(*=======================================================*)
	INIT:	(* Initialisierung *)
		st_ctrl_out.b_fehler := FALSE;
		st_ctrl_out.b_fertig := FALSE;
		st_ctrl_out.b_bereit := FALSE;
		fb_add_route_entry.bExecute := FALSE;
		fb_enum_route_entry.bExecute := FALSE;
		fb_enum_route_entry.eCmd := eEnumCmd_First;
		b_routing_station_gefunden := TRUE;
		i16_eintrag := 0;
		fb_get_local_ams_netid.bExecute := FALSE;
		fb_get_local_ams_netid.bQuit := FALSE;
		fb_get_adapters_info.bExecute := FALSE;
		fb_get_adapters_info.bQuit := FALSE;
		fb_get_host_name.bExecute := FALSE;
		fb_get_host_addr_by_name.bExecute := FALSE;
		sm_fehler_netid := FALSE;
		sm_fehler_adapter_info := FALSE;
		sm_fehler_host_name := FALSE;
		sm_fehler_host_addr := FALSE;

		FOR i16_eintrag := 0  TO (SIZEOF (arr_read_routing_info) / SIZEOF (arr_read_routing_info[0])) BY 1DO
			IF	i16_eintrag <32 THEN
				arr_read_routing_info[i16_eintrag].sName := '';
				arr_read_routing_info[i16_eintrag].sNetID := '';
				arr_read_routing_info[i16_eintrag].sAddress := '';
				arr_read_routing_info[i16_eintrag].eTransport := eRouteTransport_TCP_IP;
			END_IF
		END_FOR

		IF fb_get_local_ams_netid.bReady AND fb_get_adapters_info.bReady THEN
			fb_state_entry.i16_next_step := 20;
		END_IF

(*=======================================================*)
	20:	(* Die AMS-NetID des lokalen PC ermitteln *)
		IF fb_state_entry.E THEN
			fb_get_local_ams_netid.bExecute := TRUE;
		END_IF

		IF fb_get_local_ams_netid.bBusy THEN
			fb_get_local_ams_netid.bExecute := FALSE;
			fb_state_entry.i16_next_step := 20;
		END_IF

(*=======================================================*)
	30:
		IF NOT fb_get_local_ams_netid.bBusy  AND fb_get_local_ams_netid.bReady THEN
			IF NOT fb_get_local_ams_netid.bError THEN
				fb_state_entry.i16_next_step := 40;
			ELSE	(* Fehler *)
				sm_fehler_netid := TRUE;
				fb_state_entry.i16_next_step := 1000;
			END_IF
		END_IF

(*=======================================================*)
	40:	(* Ersten Routing Eintrag im Routingtable lesen *)
		IF fb_state_entry.E THEN
			s_temp_string_p11 := MID(fb_get_local_ams_netid.local_ams_netid, 1, 11);
			s_temp_string_p12 := MID(fb_get_local_ams_netid.local_ams_netid, 1, 12);
			s_temp_string_p13 := MID(fb_get_local_ams_netid.local_ams_netid, 1, 13);
			IF s_temp_string_p11 = '.' THEN
				(* Die vierte Zahl ist einstellig *)
				i16_temp_net_int := STRING_TO_INT(MID(fb_get_local_ams_netid.local_ams_netid, 1, 10));
			ELSIF s_temp_string_p12 = '.' THEN
				(* Die vierte Zahl ist zweistellig *)
				i16_temp_net_int := STRING_TO_INT(MID(fb_get_local_ams_netid.local_ams_netid, 2, 10));
			ELSIF s_temp_string_p13 = '.' THEN
				(* Die vierte Zahl ist dreistellig *)
				i16_temp_net_int := STRING_TO_INT(MID(fb_get_local_ams_netid.local_ams_netid, 3, 10));
			END_IF
			i16_temp_net_int := i16_temp_net_int  + 1;	(* Die NetID des Remote-Panel ist um 1 höher, als diejenige des PCs *)
			s_temp_net_string := INT_TO_STRING (i16_temp_net_int);
			s_backpanel_netid := CONCAT((CONCAT(MID(fb_get_local_ams_netid.s_ams_netid, 9, 1), s_temp_net_string)), '.1.1');
			fb_state_entry.i16_next_step := 50;
		END_IF

(*=======================================================*)
	50:	(* Die Adapter-Info des lokalen PC ermitteln *)
		IF fb_state_entry.E THEN
			fb_get_adapters_info.sNet_ID := fb_get_local_ams_netid.local_ams_netid;
			fb_get_adapters_info.bExecute := TRUE;
		END_IF

		IF fb_get_adapters_info.bBusy THEN
			fb_get_adapters_info.bExecute := FALSE;
			fb_state_entry.i16_next_step := 60;
		END_IF

(*=======================================================*)
	60:	(* Info steht zur Verfügung *)
		IF NOT fb_get_adapters_info.bBusy THEN
			IF NOT fb_get_adapters_info.bError THEN
				IF fb_get_adapters_info.bReady THEN
					st_pc_adapter_info := fb_get_adapters_info.st_ip_adapter_info;
					fb_state_entry.i16_next_step := 70;
				END_IF
			ELSE	(* Fehler *)
				sm_fehler_adapter_info := TRUE;
				fb_state_entry.i16_next_step := 1000;
			END_IF
		END_IF

(*=======================================================*)
	70:	(* Die Adapter-Info des Backpanel ermitteln *)
		IF fb_state_entry.E THEN
			fb_get_adapters_info.sNet_ID := s_backpanel_netid;
			fb_get_adapters_info.bExecute := TRUE;
		END_IF

		IF fb_get_adapters_info.bBusy THEN
			fb_get_adapters_info.bExecute := FALSE;
			fb_state_entry.i16_next_step := 80;
		END_IF

(*=======================================================*)
	80:	(* Info steht zur Verfügung *)
		IF NOT fb_get_adapters_info.bBusy THEN
			IF NOT fb_get_adapters_info.bError THEN
				IF fb_get_adapters_info.bReady THEN
					st_pc_adapter_info := fb_get_adapters_info.st_ip_adapter_info;
					s_backpanel_adresse := st_pc_adapter_info.sIpAddr;
					fb_state_entry.i16_next_step := 90;
				END_IF
			ELSE	(* Fehler *)
				sm_fehler_adapter_info := TRUE;
				fb_state_entry.i16_next_step := 1000;
			END_IF
		END_IF

(*=======================================================*)
	90:	(* Den Namen des Backpanels ermitteln *)
		IF fb_state_entry.E THEN
			fb_get_host_name.sNetID := s_backpanel_netid;
			fb_get_host_name.bExecute := TRUE;
		END_IF

		IF fb_get_host_name.bBusy THEN
			fb_get_host_name.bExecute := FALSE;
			fb_state_entry.i16_next_step := 100;
		END_IF

(*=======================================================*)
	100:	(* Info steht zur Verfügung *)
		IF NOT fb_get_host_name.bBusy THEN
			IF NOT fb_get_host_name.bError THEN
				s_backpanel_name := fb_get_host_name.sHostName;
				fb_state_entry.i16_next_step := 110;
			ELSE	(* Fehler *)
				sm_fehler_host_name := TRUE;
				fb_state_entry.i16_next_step := 1000;
			END_IF
		END_IF

(*=======================================================*)
	110:	(* Ersten Routing Eintrag im Routingtable lesen *)
		IF fb_state_entry.E THEN
			fb_enum_route_entry.bExecute := TRUE;
		END_IF

		IF fb_enum_route_entry.bBusy THEN
			fb_enum_route_entry.bExecute := FALSE;
			fb_state_entry.i16_next_step := 120;
		END_IF

(*=======================================================*)
	120:	(* Routinginformation ist vorhanden *)
		IF NOT fb_enum_route_entry.bBusy  THEN
			IF NOT fb_enum_route_entry.bError THEN
				IF NOT fb_enum_route_entry.bEOE THEN
					arr_read_routing_info[i16_eintrag] := fb_enum_route_entry.stRoute;
					fb_enum_route_entry.eCmd := eEnumCmd_Next;
					i16_eintrag := i16_eintrag + 1;
					fb_state_entry.i16_next_step := 110;
				ELSE	(* Alle vorhandenen Routingeinträge  wurden eingelesen*)
					fb_state_entry.i16_next_step := 130;
				END_IF
			ELSE	(* Fehler *)
				fb_state_entry.i16_next_step := 1000;
			END_IF
		END_IF

(*=======================================================*)
	130:	(* Alle Einträge sind gelesen *)
		IF fb_state_entry.E THEN
			(* Suche nach dem zugehörigen Backpanel *)
			FOR i16_eintrag := 0  TO (SIZEOF (arr_read_routing_info) / SIZEOF (arr_read_routing_info[0])) BY 1DO
				IF arr_read_routing_info[i16_eintrag].sNetID = s_backpanel_netid AND arr_read_routing_info[i16_eintrag].sAddress = s_backpanel_adresse THEN
					b_routing_station_gefunden := TRUE;
					fb_state_entry.i16_next_step :=  999;	(* Ende *)
					EXIT;
				ELSE
					b_routing_station_gefunden := FALSE;
				END_IF
			END_FOR
			IF NOT b_routing_station_gefunden THEN
				(* Station nicht in Liste -> eintragen *)
				fb_state_entry.i16_next_step := 140;
			END_IF
		END_IF

(*=======================================================*)
	140:	(* Routingtable mit Backpaneladresse füllen *)
		IF fb_state_entry.E THEN
			(* Initialisierung der Routingverbindung zum Backpanel *)
			fb_add_route_entry.stRoute.sName := s_backpanel_name;
			fb_add_route_entry.stRoute.sNetID := s_backpanel_netid;
			fb_add_route_entry.stRoute.sAddress := s_backpanel_adresse;
			fb_add_route_entry.stRoute.eTransport := eRouteTransport_TCP_IP;
			fb_add_route_entry.bExecute :=TRUE;
		END_IF

		IF fb_add_route_entry.bBusy THEN
			fb_add_route_entry.bExecute := FALSE;
			fb_state_entry.i16_next_step := 150;
		END_IF

(*=======================================================*)
	150:	(* Routingtable füllen läuft *)
		IF NOT fb_add_route_entry.bBusy THEN
			IF NOT fb_add_route_entry.bError THEN	(* Route wurde erfolgreich hinzugefügt *)
				fb_state_entry.i16_next_step := 999;
			ELSE	(* Fehler *)
				fb_state_entry.i16_next_step := 1000;
			END_IF
		END_IF

(*=======================================================*)
	999: (* Ende: Alle Stationen wurden im Routingtable eingetragen *)
		IF fb_r_trig_ibn_start_routing.Q THEN
			fb_state_entry.i16_next_step := INIT;
		END_IF

(*=======================================================*)
	1000: (* Fehler *)
		IF fb_state_entry.E THEN
			st_ctrl_out.b_fehler := TRUE;
			fb_ton_quitt.IN := FALSE;
			fb_add_route_entry.bExecute := FALSE;
			fb_enum_route_entry.bExecute := FALSE;
			fb_get_local_ams_netid.bExecute := FALSE;
			fb_get_local_ams_netid.bQuit := FALSE;
			fb_get_adapters_info.bExecute := FALSE;
			fb_get_adapters_info.bQuit := FALSE;
			fb_get_host_name.bExecute := FALSE;
			fb_get_host_addr_by_name.bExecute := FALSE;
		END_IF

		(*-----------------------Weiterschaltbedingungen----------------------------*)
		IF st_ctrl_in.b_quitt AND NOT fb_state_entry.E THEN
			st_ctrl_out.b_fehler := FALSE;
			fb_get_local_ams_netid .bQuit := TRUE;
			fb_get_adapters_info .bQuit := TRUE;
			fb_ton_quitt.IN := TRUE;
		END_IF

		IF fb_ton_quitt.Q OR  fb_r_trig_ibn_start_routing.Q THEN
			fb_ton_quitt.IN := FALSE;
			fb_state_entry.i16_next_step := INIT;
		END_IF
END_CASE

fb_state_entry(
	i16_next_step:= ,
	i16_pos:= 2,
	s_debugtext:= ,
	E=> ,
	X=> , 
	i16_step=> ,
	i16_last_step=> );

fb_get_local_ams_netid(
	bExecute:= , 
	bQuit:= , 
	bBusy=> , 
	bReady=> , 
	bError=> , 
	nErrId=> , 
	s_ams_netid=> );

fb_add_route_entry(
	sNetID:= '',
	stRoute:= ,
	bExecute:= ,
	tTimeout:= DEFAULT_ADS_TIMEOUT,
	bBusy=> ,
	bError=> ,
	nErrID=> );

fb_enum_route_entry(
	sNetID:= '',
	eCmd:= , 
	bExecute:= , 
	tTimeout:= DEFAULT_ADS_TIMEOUT,
	bBusy=> ,
	bError=> , 
	nErrID=> , 
	bEOE=> , 
	stRoute=> );

fb_get_adapters_info(
	sNet_ID:= , 
	bExecute:= , 
	bQuit:= , 
	bBusy=> ,
	bReady=> , 
	bError=> ,
	nErrId=> , 
	st_ip_adapter_info=> );

fb_get_host_name(
	sNetID:= ,
	bExecute:= , 
	tTimeout:= DEFAULT_ADS_TIMEOUT,
	bBusy=> , 
	bError=> ,
	nErrID=> , 
	sHostName=> );

fb_get_host_addr_by_name(
	sNetID:= '',
	sHostName:= ,
	bExecute:= , 
	tTimeout:= DEFAULT_ADS_TIMEOUT,
	bBusy=> , 
	bError=> , 
	nErrID=> , 
	sAddr=> , 
	arrAddr=> );

IF st_config.b_config_fertig THEN
	garr_stoermeldungen[st_config.i16_meld_startindex + 0] := sm_fehler_netid;
	garr_stoermeldungen[st_config.i16_meld_startindex + 1] := sm_fehler_adapter_info;
	garr_stoermeldungen[st_config.i16_meld_startindex + 2] := FALSE;
	garr_stoermeldungen[st_config.i16_meld_startindex + 3] := sm_fehler_host_addr;
	garr_stoermeldungen[st_config.i16_meld_startindex + 4] := FALSE;
	garr_stoermeldungen[st_config.i16_meld_startindex + 5] := FALSE;
	garr_stoermeldungen[st_config.i16_meld_startindex + 6] := FALSE;
	garr_stoermeldungen[st_config.i16_meld_startindex + 7] := FALSE;
	garr_stoermeldungen[st_config.i16_meld_startindex + 8] := FALSE;
	garr_stoermeldungen[st_config.i16_meld_startindex + 9] := FALSE;
	garr_stoermeldungen[st_config.i16_meld_startindex + 10] := FALSE;
	garr_stoermeldungen[st_config.i16_meld_startindex + 11] := FALSE;
	garr_stoermeldungen[st_config.i16_meld_startindex + 12] := FALSE;
	garr_stoermeldungen[st_config.i16_meld_startindex + 13] := FALSE;
	garr_stoermeldungen[st_config.i16_meld_startindex + 14] := FALSE;
	garr_stoermeldungen[st_config.i16_meld_startindex + 15] := FALSE;
	garr_stoermeldungen[st_config.i16_meld_startindex + 16] := FALSE;
	garr_stoermeldungen[st_config.i16_meld_startindex + 17] := FALSE;
	garr_stoermeldungen[st_config.i16_meld_startindex + 18] := FALSE;
	garr_stoermeldungen[st_config.i16_meld_startindex + 19] := FALSE;
	
	garr_betriebsmeldungen[st_config.i16_meld_startindex + 0] := FALSE;
	garr_betriebsmeldungen[st_config.i16_meld_startindex + 1] := FALSE;
	garr_betriebsmeldungen[st_config.i16_meld_startindex + 2] := FALSE;
	garr_betriebsmeldungen[st_config.i16_meld_startindex + 3] := FALSE;
	garr_betriebsmeldungen[st_config.i16_meld_startindex + 4] := FALSE;
	garr_betriebsmeldungen[st_config.i16_meld_startindex + 5] := FALSE;
	garr_betriebsmeldungen[st_config.i16_meld_startindex + 6] := FALSE;
	garr_betriebsmeldungen[st_config.i16_meld_startindex + 7] := FALSE;
	garr_betriebsmeldungen[st_config.i16_meld_startindex + 8] := FALSE;
	garr_betriebsmeldungen[st_config.i16_meld_startindex + 9] := FALSE;
	garr_betriebsmeldungen[st_config.i16_meld_startindex + 10] := FALSE;
	garr_betriebsmeldungen[st_config.i16_meld_startindex + 11] := FALSE;
	garr_betriebsmeldungen[st_config.i16_meld_startindex + 12] := FALSE;
	garr_betriebsmeldungen[st_config.i16_meld_startindex + 13] := FALSE;
	garr_betriebsmeldungen[st_config.i16_meld_startindex + 14] := FALSE;
	garr_betriebsmeldungen[st_config.i16_meld_startindex + 15] := FALSE;
	garr_betriebsmeldungen[st_config.i16_meld_startindex + 16] := FALSE;
	garr_betriebsmeldungen[st_config.i16_meld_startindex + 17] := FALSE;
	garr_betriebsmeldungen[st_config.i16_meld_startindex + 18] := FALSE;
	garr_betriebsmeldungen[st_config.i16_meld_startindex + 19] := FALSE;
END_IF
END_PROGRAM

(* POU EPT Lib/Programmbausteine/Routing/ST_GetAdaptersInfo, ST *)
FUNCTION_BLOCK ST_GetAdaptersInfo
VAR_INPUT
	sNet_ID						: T_AmsNetId;
	bExecute					: BOOL;
	bQuit						: BOOL;
END_VAR
VAR_OUTPUT
	bBusy						: BOOL;
	bReady						: BOOL;
	bError						: BOOL;
	nErrId						: UDINT;
	st_ip_adapter_info				: ST_IpAdapterInfo;
END_VAR
VAR
	fb_ton_quitt					: TON;
	fb_state_entry					: ST_StateEntry;
	fb_r_trig_execute				: R_TRIG;
	fb_get_adapters_info			: FB_GetAdaptersInfo;
	arr_adapters 					: ARRAY[0..MAX_LOCAL_ADAPTERS] OF ST_IpAdapterInfo;
END_VAR
(* Auslesen von IP-Adresse usw. des lokalen PCs *)
fb_r_trig_execute(CLK:= bExecute, Q=> );
fb_ton_quitt(IN:= , PT:= t#100ms, Q=> , ET=> );

(* =======================================Toplevel========================================== *)
IF fb_state_entry.i16_next_step > INIT AND fb_state_entry.i16_next_step < FEHLER THEN
	 IF fb_get_adapters_info.bError THEN
		fb_state_entry.i16_next_step := FEHLER;
	END_IF
END_IF

fb_state_entry(
	i16_next_step:= ,
	i16_pos:= 1,
	s_debugtext:= ,
	E=> ,
	X=> ,
	i16_step=> ,
	i16_last_step=> );

CASE fb_state_entry.i16_step OF
(*=======================================================*)
	0:
		fb_state_entry.i16_next_step := INIT;

(*=======================================================*)
	INIT:(* INIT *)
		bBusy := FALSE;
		bReady := FALSE;
		bError := FALSE;
		nErrId := 0;
		fb_get_adapters_info.bExecute := FALSE;
		fb_state_entry.i16_next_step := 20;

(*=======================================================*)
	20:	(* Warte auf Execute-Befehl *)
		IF fb_state_entry.E THEN
			bReady := TRUE;
		END_IF

		(*-----------------------Weiterschaltbedingungen----------------------------*)
		IF fb_r_trig_execute.Q THEN
			bReady := FALSE;
			bBusy := TRUE;
			fb_state_entry.i16_next_step := 30;
		END_IF

(*=======================================================*)
	30:	(* Starte mit Auslesen der Adapter-Info des lokalen PC *)
		IF fb_state_entry.E THEN
			fb_get_adapters_info.bExecute := TRUE;
		END_IF

		IF fb_get_adapters_info.bBusy THEN
			fb_get_adapters_info.bExecute := FALSE;
			fb_state_entry.i16_next_step := 40;
		END_IF

(*=======================================================*)
	40:	(* Adapter-Info wurde ausgelesen *)
		IF NOT fb_get_adapters_info.bBusy THEN
			IF NOT fb_get_adapters_info.bError THEN
				bBusy := FALSE;
				fb_state_entry.i16_next_step := 999;
			ELSE	(* Fehler *)
				fb_state_entry.i16_next_step := 1000;
			END_IF
		END_IF

(*=======================================================*)
	999:	(* Fertig *)
		st_ip_adapter_info := arr_adapters[1];
		fb_state_entry.i16_next_step := 20;

(*=======================================================*)
	FEHLER: (* Fehler *)
		IF fb_state_entry.E THEN
			bBusy := FALSE;
			bReady := FALSE;
			bError := TRUE;
			fb_get_adapters_info.bExecute := FALSE;
			fb_ton_quitt.IN := FALSE;
		END_IF

		(*-----------------------Weiterschaltbedingungen----------------------------*)
		IF bQuit AND NOT fb_state_entry.E THEN
			bError := FALSE;
			fb_ton_quitt.IN := TRUE;
			(* Quittierflanke für FB *)
			fb_get_adapters_info.bExecute := TRUE;
		END_IF

		IF fb_ton_quitt.Q THEN
			fb_ton_quitt.IN := FALSE;
			fb_state_entry.i16_next_step := INIT;
		END_IF
END_CASE

fb_state_entry(
	i16_next_step:= , 
	i16_pos:= 2,
	s_debugtext:= ,
	E=> ,
	X=> ,
	i16_step=> ,
	i16_last_step=> );

fb_get_adapters_info(
	sNetID:= sNet_ID,
	bExecute:= , 
	tTimeout:= DEFAULT_ADS_TIMEOUT,
	bBusy=> ,
	bError=> , 
	nErrID=> nErrId,
	arrAdapters=> arr_adapters,
	nCount=> , 
	nGet=> );
END_FUNCTION_BLOCK

(* POU EPT Lib/Programmbausteine/Routing/PC-Suche/ST_RoutingNachbarPC, ST *)
PROGRAM ST_RoutingNachbarPC
VAR_INPUT
	st_config						: struct_config;
	st_ctrl_in						: struct_ctrl_in;
END_VAR
VAR_OUTPUT
	st_ctrl_out					: struct_ctrl_out;
END_VAR
VAR
	arr_read_routing_info			: ARRAY [0..31] OF ST_AmsRouteEntry;
	fb_add_route_entry			: FB_AddRouteEntry;
	fb_enum_route_entry			: FB_EnumRouteEntry;
	fb_ton_quitt					: TON;
	fb_state_entry					: ST_StateEntry;
	i16_geschriebene_eintraege	: INT := 0;
	i16_vorhandene_eintraege		: INT := 0;
	b_ibn_start_routing			: BOOL := FALSE;
	fb_r_trig_ibn_start_routing		: R_TRIG;
	fb_ton_ibn_start_routing		: TON;
	sm_fehler_remotesuche		: BOOL := FALSE;
	sm_fehler_netid				: BOOL := FALSE;
	fb_suche_remote_pc			: ST_SucheRemotePC;
	fb_get_local_ams_netid		: ST_GetLocalAMSNetID;
	i16_eintrag					: INT := 0;
END_VAR
fb_ton_quitt(IN:= , PT:= t#100ms, Q=> , ET=> );
fb_r_trig_ibn_start_routing(CLK:= b_ibn_start_routing, Q=> );
fb_ton_ibn_start_routing(IN:= , PT:= t#1s, Q=> , ET=> );

IF fb_r_trig_ibn_start_routing.Q THEN
	fb_ton_ibn_start_routing.IN := TRUE;
ELSE
	IF fb_ton_ibn_start_routing.Q THEN
		b_ibn_start_routing := FALSE;
	 	fb_ton_ibn_start_routing.IN := FALSE;
	END_IF
END_IF

fb_state_entry(
	i16_next_step:= ,
	i16_pos:= 1,
	s_debugtext:= ,
	E=> ,
	X=> ,
	i16_step=> ,
	i16_last_step=> );

CASE fb_state_entry.i16_step OF
(*=======================================================*)
	0:	(* Initialisierung *)
		st_ctrl_out.b_fehler := TRUE;
		st_ctrl_out.b_bereit := TRUE;
		st_ctrl_out.b_fertig := TRUE;
		fb_add_route_entry.bExecute := FALSE;
		fb_enum_route_entry.bExecute := FALSE;
		fb_suche_remote_pc.bQuit := FALSE;
		fb_suche_remote_pc.bExecute := FALSE;
		fb_get_local_ams_netid .bQuit := FALSE;
		fb_get_local_ams_netid.bExecute := FALSE;
		fb_enum_route_entry.eCmd := eEnumCmd_First;
		i16_geschriebene_eintraege := 0;
		i16_vorhandene_eintraege := 0;
		sm_fehler_remotesuche := FALSE;
		sm_fehler_netid := FALSE;

		FOR i16_eintrag := 0  TO (SIZEOF (arr_read_routing_info) / SIZEOF (arr_read_routing_info[0])) BY 1DO
			arr_read_routing_info[i16_eintrag].sName := '';
			arr_read_routing_info[i16_eintrag].sNetID := '';
			arr_read_routing_info[i16_eintrag].sAddress := '';
			arr_read_routing_info[i16_eintrag].eTransport := eRouteTransport_TCP_IP;
		END_FOR

		fb_state_entry.i16_next_step := 10;

(*=======================================================*)
	10:	(* Die AMS-NetID des lokalen PC ermitteln *)
		IF fb_state_entry.E THEN
			fb_get_local_ams_netid.bExecute := TRUE;
		END_IF

		IF fb_get_local_ams_netid.bBusy THEN
			fb_get_local_ams_netid.bExecute := FALSE;
			fb_state_entry.i16_next_step := 20;
		END_IF

(*=======================================================*)
	20:
		IF NOT fb_get_local_ams_netid.bBusy  THEN
			IF NOT fb_get_local_ams_netid.bError THEN
				fb_state_entry.i16_next_step := 100;
			ELSE	(* Fehler *)
				sm_fehler_netid := TRUE;
				fb_state_entry.i16_next_step := 1000;
			END_IF
		END_IF

(*=======================================================*)
	100:	(* Ersten Routing Eintrag im Routingtable lesen *)
		IF fb_state_entry.E THEN
			fb_enum_route_entry.bExecute := TRUE;
		END_IF

		IF fb_enum_route_entry.bBusy THEN
			fb_enum_route_entry.bExecute := FALSE;
			fb_state_entry.i16_next_step := 110;
		END_IF

(*=======================================================*)
	110:	(* Routinginformation ist vorhanden *)
		IF NOT fb_enum_route_entry.bBusy  THEN
			IF NOT fb_enum_route_entry.bError THEN
				IF NOT fb_enum_route_entry.bEOE THEN
					arr_read_routing_info[i16_vorhandene_eintraege] := fb_enum_route_entry.stRoute;
					fb_enum_route_entry.eCmd := eEnumCmd_Next;
					fb_state_entry.i16_next_step := 120;
				ELSE	(* Alle vorhandenen Routingeinträge  wurden eingelesen*)
					fb_state_entry.i16_next_step := 130;
				END_IF
			ELSE	(* Fehler *)
				fb_state_entry.i16_next_step := 1000;
			END_IF
		END_IF

(*=======================================================*)
	120:	(* Zähler erhöhen *)
		IF fb_state_entry.E THEN
			i16_vorhandene_eintraege := i16_vorhandene_eintraege + 1;
		END_IF

		fb_state_entry.i16_next_step := 100;

(*=======================================================*)
	130:	(* Suche Nachbar-PCs im Maschinennetz *)
		IF fb_state_entry.E THEN
			fb_suche_remote_pc.bExecute := TRUE;
		END_IF

		IF fb_suche_remote_pc.bBusy THEN
			fb_suche_remote_pc.bExecute := FALSE;
			fb_state_entry.i16_next_step := 140;
		END_IF

(*=======================================================*)
	140:	(* Suchvorgang und beendet *)
		IF NOT fb_suche_remote_pc.bBusy  THEN
			IF NOT fb_suche_remote_pc.bError THEN
				fb_state_entry.i16_next_step := 150;
			ELSE	(* Fehler *)
				sm_fehler_remotesuche := TRUE;
				fb_state_entry.i16_next_step := 1000;
			END_IF
		END_IF

(*=======================================================*)
	150:	(* Die Route der gefundenen Nachbar-PCs eintragen *)
		IF fb_state_entry.E THEN
			fb_add_route_entry.stRoute.sName := fb_suche_remote_pc.st_remote_pcinfo_struct[i16_geschriebene_eintraege].Name;
			fb_add_route_entry.stRoute.sNetID := fb_suche_remote_pc.st_remote_pcinfo_struct[i16_geschriebene_eintraege].NetId;
			fb_add_route_entry.stRoute.sAddress := DELETE(fb_add_route_entry.stRoute.sNetID, 4, 12);
			fb_add_route_entry.stRoute.eTransport := eRouteTransport_TCP_IP;
			fb_add_route_entry.bExecute :=TRUE;
			i16_geschriebene_eintraege := i16_geschriebene_eintraege + 1;
		END_IF

		IF fb_add_route_entry.bBusy THEN
			fb_add_route_entry.bExecute := FALSE;
			fb_state_entry.i16_next_step := 160;
		END_IF

(*=======================================================*)
	160:	(* Routingtable füllen läuft *)
		IF NOT fb_add_route_entry.bBusy THEN
			IF NOT fb_add_route_entry.bError THEN	(* Route wurde erfolgreich hinzugefügt *)
				(* Routingtable mit fehlenden Stationsadressen füllen wenn notwendig *)
				IF i16_geschriebene_eintraege < i16_vorhandene_eintraege THEN
					fb_state_entry.i16_next_step := 150;
				ELSE
					fb_state_entry.i16_next_step := 999;
				END_IF
			ELSE	(* Fehler *)
				fb_state_entry.i16_next_step := 1000;
			END_IF
		END_IF

(*=======================================================*)
	999: (* Ende: Alle Stationen wurden im Routingtable eingetragen *)
		IF fb_state_entry.E THEN
			st_ctrl_out.b_fertig := TRUE;
		END_IF

(*=======================================================*)
	1000: (* Fehler *)
		IF fb_state_entry.E THEN
			st_ctrl_out.b_fehler := TRUE;
			fb_ton_quitt.IN := FALSE;
			fb_add_route_entry.bExecute := FALSE;
			fb_enum_route_entry.bExecute := FALSE;
			fb_suche_remote_pc.bExecute := FALSE;
			fb_suche_remote_pc.bQuit := FALSE;
			fb_get_local_ams_netid.bExecute := FALSE;
			fb_get_local_ams_netid.bQuit := FALSE;
		END_IF

		(*-----------------------Weiterschaltbedingungen----------------------------*)
		IF st_ctrl_in.b_quitt AND NOT fb_state_entry.E THEN
			st_ctrl_out.b_fehler := FALSE;
			fb_ton_quitt.IN := TRUE;
			fb_suche_remote_pc.bQuit := TRUE;
			fb_get_local_ams_netid .bQuit := TRUE;
		END_IF

		IF fb_ton_quitt.Q OR  fb_r_trig_ibn_start_routing.Q THEN
			fb_ton_quitt.IN := FALSE;
			fb_state_entry.i16_next_step := 0;
		END_IF
END_CASE

fb_state_entry(
	i16_next_step:= , 
	i16_pos:= 2,
	s_debugtext:= ,
	E=> ,
	X=> , 
	i16_step=> ,
	i16_last_step=> );

fb_get_local_ams_netid(
	bExecute:= , 
	bQuit:= , 
	bBusy=> , 
	bReady=> , 
	bError=> , 
	nErrId=> , 
	s_ams_netid=> );

fb_suche_remote_pc(
	bExecute:= ,
	bQuit:= , 
	bBusy=> , 
	bError=> , 
	nErrId=> );

fb_add_route_entry(
	sNetID:= ,
	stRoute:= ,
	bExecute:= ,
	tTimeout:= DEFAULT_ADS_TIMEOUT,
	bBusy=> , 
	bError=> , 
	nErrID=> );

fb_enum_route_entry(
	sNetID:= ,
	eCmd:= , 
	bExecute:= , 
	tTimeout:= DEFAULT_ADS_TIMEOUT,
	bBusy=> , 
	bError=> , 
	nErrID=> , 
	bEOE=> , 
	stRoute=> );

IF st_config.b_config_fertig THEN
	garr_stoermeldungen[st_config.i16_meld_startindex + 0] := sm_fehler_remotesuche;
	garr_stoermeldungen[st_config.i16_meld_startindex + 1] := sm_fehler_netid;
	garr_stoermeldungen[st_config.i16_meld_startindex + 2] := FALSE;
	garr_stoermeldungen[st_config.i16_meld_startindex + 3] := FALSE;
	garr_stoermeldungen[st_config.i16_meld_startindex + 4] := FALSE;
	garr_stoermeldungen[st_config.i16_meld_startindex + 5] := FALSE;
	garr_stoermeldungen[st_config.i16_meld_startindex + 6] := FALSE;
	garr_stoermeldungen[st_config.i16_meld_startindex + 7] := FALSE;
	garr_stoermeldungen[st_config.i16_meld_startindex + 8] := FALSE;
	garr_stoermeldungen[st_config.i16_meld_startindex + 9] := FALSE;
	garr_stoermeldungen[st_config.i16_meld_startindex + 10] := FALSE;
	garr_stoermeldungen[st_config.i16_meld_startindex + 11] := FALSE;
	garr_stoermeldungen[st_config.i16_meld_startindex + 12] := FALSE;
	garr_stoermeldungen[st_config.i16_meld_startindex + 13] := FALSE;
	garr_stoermeldungen[st_config.i16_meld_startindex + 14] := FALSE;
	garr_stoermeldungen[st_config.i16_meld_startindex + 15] := FALSE;
	garr_stoermeldungen[st_config.i16_meld_startindex + 16] := FALSE;
	garr_stoermeldungen[st_config.i16_meld_startindex + 17] := FALSE;
	garr_stoermeldungen[st_config.i16_meld_startindex + 18] := FALSE;
	garr_stoermeldungen[st_config.i16_meld_startindex + 19] := FALSE;
	
	garr_betriebsmeldungen[st_config.i16_meld_startindex + 0] := FALSE;
	garr_betriebsmeldungen[st_config.i16_meld_startindex + 1] := FALSE;
	garr_betriebsmeldungen[st_config.i16_meld_startindex + 2] := FALSE;
	garr_betriebsmeldungen[st_config.i16_meld_startindex + 3] := FALSE;
	garr_betriebsmeldungen[st_config.i16_meld_startindex + 4] := FALSE;
	garr_betriebsmeldungen[st_config.i16_meld_startindex + 5] := FALSE;
	garr_betriebsmeldungen[st_config.i16_meld_startindex + 6] := FALSE;
	garr_betriebsmeldungen[st_config.i16_meld_startindex + 7] := FALSE;
	garr_betriebsmeldungen[st_config.i16_meld_startindex + 8] := FALSE;
	garr_betriebsmeldungen[st_config.i16_meld_startindex + 9] := FALSE;
	garr_betriebsmeldungen[st_config.i16_meld_startindex + 10] := FALSE;
	garr_betriebsmeldungen[st_config.i16_meld_startindex + 11] := FALSE;
	garr_betriebsmeldungen[st_config.i16_meld_startindex + 12] := FALSE;
	garr_betriebsmeldungen[st_config.i16_meld_startindex + 13] := FALSE;
	garr_betriebsmeldungen[st_config.i16_meld_startindex + 14] := FALSE;
	garr_betriebsmeldungen[st_config.i16_meld_startindex + 15] := FALSE;
	garr_betriebsmeldungen[st_config.i16_meld_startindex + 16] := FALSE;
	garr_betriebsmeldungen[st_config.i16_meld_startindex + 17] := FALSE;
	garr_betriebsmeldungen[st_config.i16_meld_startindex + 18] := FALSE;
	garr_betriebsmeldungen[st_config.i16_meld_startindex + 19] := FALSE;
END_IF
END_PROGRAM

(* POU EPT Lib/Programmbausteine/Routing/PC-Suche/ST_SucheRemotePC, ST *)
FUNCTION_BLOCK ST_SucheRemotePC
VAR_INPUT
	bExecute			: BOOL;
	bQuit				: BOOL;
END_VAR
VAR_OUTPUT
	bBusy				: BOOL;
	bError				: BOOL;
	nErrId				: UDINT;
END_VAR
VAR
	fb_ton_quitt					: TON;
	fb_state_entry					: ST_StateEntry;
	fb_r_trig_execute				: R_TRIG;
	i							: INT := 0;
	b_ibn_start					: BOOL := FALSE;
	fb_r_trig_ibn_start				: R_TRIG;
	fb_ton_ibn_start				: TON;
	fb_get_remote_pcinfo			:GetRemotePCInfo;
	st_remote_pcinfo_struct		:REMOTEPCINFOSTRUCT;
							       (*TYPE REMOTEPCINFOSTRUCT
									ARRAY[0..99] OF REMOTEPC;
								END_TYPE*)
							      (*TYPE REMOTEPC
								STRUCT
									NetId 	: T_AmsNetId;
									Name 	: STRING(31);
								END_STRUCT
								END_TYPE*)
END_VAR
fb_r_trig_execute(CLK:= bExecute, Q=> );
fb_ton_quitt(IN:= , PT:= t#100ms, Q=> , ET=> );

fb_r_trig_ibn_start(CLK:= b_ibn_start, Q=> );
fb_ton_ibn_start(IN:= , PT:= t#1s, Q=> , ET=> );

IF fb_r_trig_ibn_start.Q THEN
	fb_ton_ibn_start.IN := TRUE;
ELSE
	IF fb_ton_ibn_start.Q THEN
		b_ibn_start := FALSE;
	 	fb_ton_ibn_start.IN := FALSE;
	END_IF
END_IF

fb_state_entry(
	i16_next_step:= ,
	i16_pos:= 1,
	s_debugtext:= ,
	E=> ,
	X=> , 
	i16_step=> ,
	i16_last_step=> );

CASE fb_state_entry.i16_step OF
(*=======================================================*)
	0:(* INIT *)
		bBusy := FALSE;
		bError := FALSE;
		nErrId := 0;
		fb_get_remote_pcinfo.START := FALSE;
		fb_state_entry.i16_next_step := 10;

(*=======================================================*)
	10:	(* Warte auf Execute-Befehl *)
		IF fb_state_entry.E THEN
			bBusy := FALSE;
		END_IF

		IF fb_r_trig_execute.Q OR fb_r_trig_ibn_start.Q THEN
			bBusy := TRUE;
			fb_state_entry.i16_next_step := 100;
		END_IF

(*=======================================================*)
	100:	(* Starte mit Auslesen der über ADS verbundenen Nachbar-PCs *)
		IF fb_state_entry.E THEN
			fb_get_remote_pcinfo.START := TRUE;
		END_IF

		IF fb_get_remote_pcinfo.BUSY THEN
			fb_get_remote_pcinfo.START := FALSE;
			fb_state_entry.i16_next_step := 110;
		END_IF

(*=======================================================*)
	110:	(* Routinginformation über die Nachbar-PCs ist vorhanden *)
		IF NOT fb_get_remote_pcinfo.BUSY  THEN
			IF NOT fb_get_remote_pcinfo.ERR THEN
				fb_state_entry.i16_next_step := 999;
			ELSE	(* Fehler *)
				fb_state_entry.i16_next_step := 1000;
			END_IF
		END_IF

(*=======================================================*)
	999:	(* Kontrollschritt: Nachbar-PC ist gefunden *)
		fb_state_entry.i16_next_step := 10;

(*=======================================================*)
	1000: (* Fehler *)
		IF fb_state_entry.E THEN
			bBusy := FALSE;
			bError := TRUE;
			fb_ton_quitt.IN := FALSE;
		END_IF

		(*-----------------------Weiterschaltbedingungen----------------------------*)
		IF bQuit AND NOT fb_state_entry.E THEN
			bError := FALSE;
			fb_ton_quitt.IN := TRUE;
		END_IF

		IF fb_ton_quitt.Q THEN
			fb_ton_quitt.IN := FALSE;
			fb_state_entry.i16_next_step := 0;
		END_IF
END_CASE

fb_state_entry(
	i16_next_step:= , 
	i16_pos:= 2,
	s_debugtext:= ,
	E=> ,
	X=> , 
	i16_step=> ,
	i16_last_step=> );

fb_get_remote_pcinfo(
	NETID:= , 
	START:= , 
	TMOUT:= , 
	BUSY=> , 
	ERR=> , 
	ERRID=> , 
	RemotePCInfo=> st_remote_pcinfo_struct);
END_FUNCTION_BLOCK

(* POU EPT Lib/Programmbausteine/ST_start_OSK, ST *)
PROGRAM ST_start_OSK
VAR_INPUT
	bExecute			: BOOL;
END_VAR
VAR
	NT_StartProcess 		:NT_StartProcess;
	b_Start				:BOOL;

	fb_ton_start			:TON;
	fb_r_trig_start			: R_TRIG;

END_VAR
(*Windows Tastatur starten mit der Quttiertaste*)
fb_ton_start(
	IN:=bExecute,
	PT:= t#2s,);

fb_r_trig_start(
	CLK:=fb_ton_start.Q ,
	Q=> b_Start);

NT_StartProcess(
	NETID:='',
	PATHSTR	:='C:\Windows\System32\cmd.exe',
	DIRNAME	:= ,
	COMNDLINE	:='/C C:\WINDOWS\system32\taskkill /f /im osk.exe /t & start /b osk /MAX',
	START		:=b_Start,
	TMOUT		:=T#10s);

IF	NOT NT_StartProcess.BUSY AND b_Start THEN
	b_Start:=FALSE;
END_IF
END_PROGRAM

(* POU EPT Lib/Programmbausteine/ST_System_DateAndTime, ST *)
PROGRAM ST_System_DateAndTime
VAR
	w_year					: WORD := 16#0000;
	w_month					: WORD := 16#0000;
	w_day					: WORD := 16#0000;
	w_hour					: WORD := 16#0000;
	w_min					: WORD := 16#0000;
	w_sec					: WORD := 16#0000;
	fb_get_system_time 		: FB_LocalSystemTime;
END_VAR
(* =====Erzeugen der Systemzeit für die ganze Maschine======== *)
(* Die Umstellung von Sommer auf Winterzeit und umgekehrt erfolgt automatisch über die PC-Zeit *)
fb_get_system_time ( sNetID := '',
					bEnable 	:= TRUE,
					dwCycle 	:= 1,
					dwOpt	:= 1,
					tTimeout 	:= DEFAULT_ADS_TIMEOUT,
					bValid => b_system_time_valid,
					systemTime => gst_system_time, (* Systemzeit *)
					tzID 	=> );
(*=======================================================*)
gdt_system_time := SYSTEMTIME_TO_DT(fb_get_system_time.systemTime);

w_year:=gst_system_time.wYear;
w_month:=gst_system_time.wMonth;
w_day:=gst_system_time.wDay;
w_hour:=gst_system_time.wHour;
w_min:=gst_system_time.wMinute;
w_sec:=gst_system_time.wSecond;

gstr_system_time := '';
gstr_datum := '';
IF w_day < 10 THEN
	gstr_datum := CONCAT(gstr_datum ,WORD_TO_STRING(0));
END_IF;
gstr_datum := CONCAT(gstr_datum ,WORD_TO_STRING(w_day));
gstr_datum := CONCAT(gstr_datum , '.');

IF w_month < 10 THEN
	gstr_datum := CONCAT(gstr_datum ,WORD_TO_STRING(0));
END_IF;
gstr_datum := CONCAT(gstr_datum ,WORD_TO_STRING(w_month));
gstr_datum := CONCAT(gstr_datum , '.');
gstr_datum := CONCAT(gstr_datum ,WORD_TO_STRING(w_year));	(* Datum steht zur Verfügung *)

gstr_uhrzeit := '';
IF w_hour < 10 THEN
	gstr_uhrzeit := CONCAT(gstr_uhrzeit ,WORD_TO_STRING(0));
END_IF;
gstr_uhrzeit := CONCAT(gstr_uhrzeit ,WORD_TO_STRING(w_hour));
gstr_uhrzeit := CONCAT(gstr_uhrzeit , ':');

IF w_min < 10 THEN
	gstr_uhrzeit := CONCAT(gstr_uhrzeit ,WORD_TO_STRING(0));
END_IF;
gstr_uhrzeit := CONCAT(gstr_uhrzeit ,WORD_TO_STRING(w_min));
gstr_uhrzeit := CONCAT(gstr_uhrzeit , ':');

IF w_sec < 10 THEN
	gstr_uhrzeit := CONCAT(gstr_uhrzeit ,WORD_TO_STRING(0));
END_IF;
gstr_uhrzeit := CONCAT(gstr_uhrzeit ,WORD_TO_STRING(w_sec));	(* Uhrzeit steht zur Verfügung *)

gstr_system_time := CONCAT(gstr_system_time, gstr_datum );
gstr_system_time := CONCAT(gstr_system_time , ' ');
gstr_system_time := CONCAT(gstr_system_time , gstr_uhrzeit);	(* Ausgabe von Datum und Uhrzeit als String für z.B . die Visu *)
END_PROGRAM

(* POU EPT Lib/Programmbausteine/ST_UPS, ST *)
PROGRAM ST_UPS
VAR_INPUT
	st_config				: struct_config;
	st_ctrl_in				: struct_ctrl_in;
	b_Ups					: BOOL;
END_VAR
VAR_IN_OUT

END_VAR
VAR_OUTPUT
	st_ctrl_out			: struct_ctrl_out;
END_VAR
VAR
	fb_ton_quitt			: TON;
	fb_ton_uez			: TON;
	fb_state_entry			: ST_StateEntry;

	nLastErrID			:UDINT;

	fbGetUpsStatus		: FB_GetUPSStatus;

	bm_ReplaceBattery 	: BOOL;
	bm_NoPower 		: BOOL;
	bm_StatusNotValid 	: BOOL;
END_VAR
(*======================================================
   ST: ST_UPS
 ------------------------------------------------------
   Auth: 	Thomas Vilgis    						 
   Date: 	21.06.2018    						     
   Rev.: 		1.0	
   Desc:		Der Baustein liest den Status des Akkupacks aus.
			Die restliche Akkulaufzeit in Minuten kann abgefragt werden.
			Wenn der Akkupack getauscht werden muss wird angezeigt.
			Wenn sich der PC im Netzbetrieb befindet wird angezeigt.
   Historie: 	1.0

 ========================================================*)

(* Zeiten *)
fb_ton_quitt(IN:= , PT:= t#100ms, Q=> , ET=> );
fb_ton_uez(IN:= , PT:= t#20s, Q=> , ET=> );

(* Flanken *)


(* Toplevel *)
IF fb_state_entry.i16_next_step > INIT AND fb_state_entry.i16_next_step < FEHLER  THEN
	IF fb_state_entry.i16_next_step < STOP THEN
		IF st_ctrl_in.b_stop THEN
			fb_state_entry.i16_next_step := STOP;
		END_IF
	END_IF
END_IF

(* ======================================Schrittkette======================================== *)
fb_state_entry(	i16_pos:= 1);

CASE fb_state_entry.i16_step OF
(*=======================================================*)
	INIT_OBJ:
		IF st_config.b_config_fertig THEN
			fb_state_entry.i16_next_step := INIT;
		END_IF

(*=======================================================*)
	INIT:
		IF fb_state_entry.E THEN
			fb_ton_quitt.IN := FALSE;
			fb_ton_uez.IN := FALSE;
			st_ctrl_out.b_fehler := FALSE;
			st_ctrl_out.b_bereit := FALSE;
			st_ctrl_out.b_fertig := FALSE;
			st_ctrl_out.b_busy := FALSE;

			bm_ReplaceBattery := FALSE;
			bm_NoPower := FALSE;
			bm_StatusNotValid := FALSE;

			fbGetUpsStatus.bEnable := FALSE;
		END_IF

		(*-----------------------Weiterschaltbedingungen----------------------------*)
		fb_state_entry.i16_next_step := BEREIT;

(*=======================================================*)
	BEREIT:
		IF fb_state_entry.E THEN
			st_ctrl_out.b_bereit := TRUE;
		END_IF

		fbGetUpsStatus.bEnable := b_Ups;
		fb_ton_uez.IN := b_Ups;

		(*-----------------------Weiterschaltbedingungen----------------------------*)
		IF b_Ups THEN
			IF fbGetUpsStatus.bValid THEN
				fb_state_entry.i16_next_step := 110;
			ELSIF fb_ton_uez.Q THEN
				bm_StatusNotValid := TRUE;
				fb_state_entry.i16_next_step := FEHLER;
			END_IF
		END_IF

		IF fb_state_entry.X THEN
			st_ctrl_out.b_bereit := FALSE;
			st_ctrl_out.b_fertig := FALSE;
			st_ctrl_out.b_busy := TRUE;
		END_IF

(*=======================================================*)
	110:	(* Evaluation *)

		(*-----------------------Weiterschaltbedingungen----------------------------*)
		IF fbGetUpsStatus.bValid THEN
			IF NOT fbGetUpsStatus.bError THEN
				CASE fbGetUpsStatus.stStatus.eBatteryStatus OF
					BatteryUnknownStatus:	(*Der Akkustatus ist unbekannt*)
						;
					BatteryOk:			(*Der Akku ist in Ordnung*)
						bm_ReplaceBattery := FALSE;
					BatteryReplace:		(*Der Akku sollte gewechselt werden*)
						bm_ReplaceBattery := TRUE;
				END_CASE

				CASE fbGetUpsStatus.stStatus.eCommStatus OF
					UpsCommUnknownStatus:	(*Kommunikationsstatus zur USV-Hardware ist unbekannt*)
						;
					UpsCommOk:		(*Kommunikation zur USV-Hardware ist hergestellt*)
						;
					UpsCommFailed:	(*Kommunikation zur USV wurde unterbrochen*)
						;
				END_CASE

				CASE fbGetUpsStatus.stStatus.ePowerStatus OF
					PowerUnknownStatus:	(*Der Status der Stromversorgung ist unbekannt*)
						;
					PowerOnLine:		(*Das Gerät befindet sich im Netzbetrieb*)
						bm_NoPower := FALSE;
					PowerOnBattery:	(*Stromausfall ist aufgetreten und das Gerät befindet sich im Akkubetrieb*)
						bm_NoPower := TRUE;
				END_CASE
			ELSE
				nLastErrID := fbGetUpsStatus.nErrId;
				fb_state_entry.i16_next_step := FEHLER;
			END_IF
		ELSE
			bm_StatusNotValid := TRUE;
			fb_state_entry.i16_next_step := FEHLER;
		END_IF

(*=======================================================*)
	STOP, FEHLER:
		IF fb_state_entry.E THEN
			st_ctrl_out.b_fehler := fb_state_entry.i16_step = FEHLER;
			st_ctrl_out.b_gestoppt := fb_state_entry.i16_step = STOP;
			fb_ton_quitt.IN := FALSE;
			fbGetUpsStatus.bEnable := FALSE;
		END_IF

		(*-----------------------Weiterschaltbedingungen----------------------------*)
		IF st_ctrl_in.b_quitt THEN
			st_ctrl_out.b_fehler := FALSE;
			fb_ton_quitt.IN := TRUE;
		END_IF
	
		IF fb_ton_quitt.Q THEN
			fb_ton_quitt.IN := FALSE;
			fb_state_entry.i16_next_step := INIT;
		END_IF

END_CASE

fb_state_entry(i16_pos:= 2 );

fbGetUpsStatus(
	sNetId:= ,	(* wenn in AmsNetId nichts drin steht, wird immer die lokale genommen*)
	nPort:= 0,
	bEnable:= ,
	bValid=> , 
	bError=> , 
	nErrId=> ,
	stStatus=> );

IF st_config.b_config_fertig THEN
	(* Fehlermeldungen und Betriebsmeldungen ab dem Startindex in die globalen Meldungsarrays schreiben *)
	garr_stoermeldungen[st_config.i16_meld_startindex + 0] := FALSE;
	garr_stoermeldungen[st_config.i16_meld_startindex + 1] := FALSE;
	garr_stoermeldungen[st_config.i16_meld_startindex + 2] := FALSE;
	garr_stoermeldungen[st_config.i16_meld_startindex + 3] := FALSE;
	garr_stoermeldungen[st_config.i16_meld_startindex + 4] := FALSE;

	garr_betriebsmeldungen[st_config.i16_meld_startindex + 0] := bm_ReplaceBattery;
	garr_betriebsmeldungen[st_config.i16_meld_startindex + 1] := bm_NoPower;
	garr_betriebsmeldungen[st_config.i16_meld_startindex + 2] := bm_StatusNotValid;
	garr_betriebsmeldungen[st_config.i16_meld_startindex + 3] := FALSE;
	garr_betriebsmeldungen[st_config.i16_meld_startindex + 4] := FALSE;
END_IF
END_PROGRAM

(* POU Gemeinsamkeiten17xx/Achsen/ST_Bestueckachse, ST *)
PROGRAM ST_Bestueckachse
VAR_INPUT
	st_config_achse						: struct_ecd_config;
	st_ctrl_in								: struct_ctrl_in;
	e_steuerung_ein						: BOOL;
	e_ba_mit_bedingungen				: BOOL;
	e_tuere_vorne_offen					: BOOL;
	e_tuere_hinten_offen					: BOOL;
END_VAR
VAR_IN_OUT
	st_visu								: struct_ecd_visu;
END_VAR
VAR_OUTPUT
	st_ctrl_out							: struct_ctrl_out;
END_VAR
VAR
	st_sm						 		: struct_ecd_meldungen;
	st_drive_cmd							: struct_ecd_cmd;
	fb_ton_wz							: TON;
	fb_ton_quitt							: TON;
	fb_ton_wz_disable						: TON;
	fb_r_trig_tippen						: R_TRIG;
	fb_f_trig_tippen						: F_TRIG;
	fb_r_trig_taste_plus					: R_TRIG;
	fb_r_trig_taste_minus					: R_TRIG;
	fb_r_trig_start							: R_TRIG;
	fb_r_trig_hand_dialog					: R_TRIG;
	fb_r_trig_nullpunkt_setzen				: R_TRIG;
	fb_axis								: ST_AxisJobCtrl_Motion;
	fb_state_entry							: ST_StateEntry;
	fb_ton_uez							: TON;
	i, j									: INT := 0;
	lr_pos_ohneverschiebung			: LREAL;
	st_geschwindigkeiten					: struct_ecd_geschwindigkeiten;
	b_hand_dialog_aktiv					: BOOL := FALSE;
	b_nullnockenmerker					: BOOL := FALSE;

	sm_fehler_initialposition_achse			: BOOL := FALSE;
	sm_keine_nocken_definiert				: BOOL := FALSE;
	sm_fehler_ot_ut						: BOOL := FALSE;

	e_referenz_sensor						AT %I* : BOOL;
	i16_torque							AT %I* : INT;

	fb_ot_ut_ueberwachung				: ST_OT_UT_Ueberwachung;

	lr_decceleration_nothalt				: LREAL;
	lr_decceleration_normal				: LREAL;
END_VAR
(* Zeiten *)
fb_ton_wz(IN:= ,PT:= , Q=>  , ET=> );
fb_ton_uez(IN:= ,	PT:= , Q=>  , ET=> );
fb_ton_quitt(IN:= , PT:= t#100ms, Q=> , ET=> );
fb_ton_wz_disable(IN:= , PT:= t#500ms, Q=> , ET=> );

(* Flanken *)
fb_r_trig_taste_plus(CLK:= ST_Euchner_Handbedienpult.b_Taste_Plus, Q=> );
fb_r_trig_taste_minus(CLK:= ST_Euchner_Handbedienpult.b_Taste_Minus, Q=> );
fb_r_trig_start(CLK:= st_ctrl_in.b_start, Q=> );
fb_r_trig_hand_dialog(CLK:= b_hand_dialog_aktiv, Q=> );
fb_r_trig_nullpunkt_setzen(CLK:= axis_bestueckachse.st_visu.b_nullpunkt_setzen, Q=> );

(* Achse steuern *)
(* Bestueckachse *)
fb_axis(
	e_referenznocken:= ,
	b_refsensor_vorhanden:= st_config_achse.b_refsensor_vorhanden,
	b_limitsensor_positiv_vorhanden:= st_config_achse.b_limitsensor_positiv_vorhanden,
	b_limitsensor_negativ_vorhanden:= st_config_achse.b_limitsensor_negativ_vorhanden,
	i16_achstyp := st_config_achse.i16_achstyp,
	st_position:= ,
	lr_override_vorgabe:= ST_TippTasten.lr_override,
	mc_richtung_modulo:= ,
	mc_richtung_velocity:= ,
	mc_referenzmodus:= ,
	mc_buffermode_axis:= ,
	ui16_soeparam_write_value:= ,
	w_idn:= ,
	i16_nc_parameter_nummer:= ,
	r_wert_nc_write_parameter:= ,
	st_vorgabe_geschwindigkeiten:= st_geschwindigkeiten,
	lr_soll_geschwindigkeit:=,
	b_bedingung_sls:= NOT e_tuere_vorne_offen OR NOT e_tuere_hinten_offen,
	st_ads_info := ,
	st_eccoe_sdo := ,
	st_masterachse:= bestueckachse,
	st_visu_axis:= st_visu,
	st_ecd_cmd:= st_drive_cmd,
	ui16_soeparam_read_value=> ,
	r_wert_nc_read_parameter=> );

IF gi16_betriebsart <> AUTO THEN
	(* Bausteinaufruf für Kontrolle der korrekten Abfolge von OT zu UT. Nicht für Automatikbetrieb geeignet, da Aufruf in der normalen Task! *)
	fb_ot_ut_ueberwachung(
		lr_achsposition:= bestueckachse.NcToPlc.ModuloActPos,
		b_error=> sm_fehler_ot_ut);
ELSE
	sm_fehler_ot_ut := FALSE;
END_IF

IF gi16_betriebsart = HAND THEN
	(* Achse mit dem Euchner Handbediengerät vorwärts und rückwärts Bewegen*)
	IF fb_r_trig_hand_dialog.Q THEN
		fb_state_entry.i16_next_step := HANDRAD;
	END_IF

	(* Button in der Oberfläche zum setzen des Nullpunktes *)
	IF fb_r_trig_nullpunkt_setzen.Q THEN
		fb_state_entry.i16_next_step :=	NULLPUNKT_SETZEN;
	END_IF
END_IF


(* =======================================Toplevel========================================== *)
(* Starte Inbetriebnahme-Sequenz *)
IF st_ctrl_in.b_gehe_step_ibn THEN
	fb_state_entry.i16_next_step := INBETRIEBNAHME;
END_IF

(* =====Achse wird disabled===== *)
IF (NOT e_steuerung_ein OR NOT e_ba_mit_bedingungen) AND bestueckachse.Status.Operational THEN
	st_drive_cmd.enu_cmd := POWER_DISABLE;
END_IF

IF fb_state_entry.i16_next_step > INIT AND fb_state_entry.i16_next_step < FEHLER THEN
	(* =====Fehler vom Achskontroller===== *)
	IF st_drive_cmd.b_job_fehler THEN
		fb_state_entry.i16_next_step := FEHLER;
	END_IF

	IF fb_state_entry.i16_next_step > 45 THEN
		(* Devicefehler *)
		IF bestueckachse.Status.Error THEN
			st_sm.b_achsfehler := TRUE;
			fb_state_entry.i16_next_step := FEHLER;
		ELSIF bestueckachse.Status.DriveDeviceError THEN
			st_sm.b_devicefehler := TRUE;
			fb_state_entry.i16_next_step := FEHLER;
		END_IF
	END_IF

	IF fb_state_entry.i16_next_step < STOP THEN
		(* =====Achse wird gestoppt===== *)
		IF st_ctrl_in.b_stop THEN
			fb_state_entry.i16_next_step := STOP;
		ELSIF fb_state_entry.i16_next_step < HALT THEN
			(* =====Achse wird angehalten===== *)
			IF st_ctrl_in.b_halt THEN
				fb_state_entry.i16_next_step := HALT;
			END_IF
		END_IF
	END_IF
END_IF

(* ======================================Schrittkette======================================== *)
fb_state_entry(
	i16_next_step:= ,
	i16_pos:= 1,
	s_debugtext:= ,
	E=> ,
	X=> ,
	i16_step=> ,
	i16_last_step=> );

CASE fb_state_entry.i16_step OF
(*=======================================================*)
	INIT_OBJ:
		IF st_config_achse.b_config_fertig THEN
			fb_state_entry.i16_next_step := 1;
		END_IF

(*=======================================================*)
	1:	(* Warte bis NetID´s der Slaves ausgelesen sind *)
		IF fb_state_entry.E THEN
			;
		END_IF

		(*-----------------------Weiterschaltbedingungen----------------------------*)
		IF ST_EthercatDiag.st_ctrl_out.b_fertig THEN
			fb_state_entry.i16_next_step := 3;
		END_IF

(*=======================================================*)
	3:	(* Spezifische NC-Achsparameter auslesen *)
		IF fb_state_entry.E THEN
			FOR i := 0  TO (SIZEOF (nockenschaltwerk_bestueckachse.fb.arr_spur) / SIZEOF (nockenschaltwerk_bestueckachse.fb.arr_spur[0])) - 1 BY 1DO
				gst_datensatz.st_wkz.nockenschaltwerk_bestueckachse.arr_nocken[i].b_camvalid := TRUE;
			END_FOR

			fb_axis.i16_nc_parameter_nummer := MaxVelocitySystem;
			st_drive_cmd.enu_cmd := READ_NC_PARAMETER;
		END_IF

		(*-----------------------Weiterschaltbedingungen----------------------------*)
		IF st_drive_cmd.enu_cmd = NO_COMMAND THEN
			st_geschwindigkeiten.lr_maximalgeschwindigkeit := fb_axis.r_wert_nc_read_parameter(* °/s *) * 60 / 360;
			st_geschwindigkeiten.lr_auto_max := st_geschwindigkeiten.lr_maximalgeschwindigkeit;
			st_geschwindigkeiten.lr_auto_min := 50;
			st_geschwindigkeiten.lr_jog := 100;
			fb_state_entry.i16_next_step := 4;
		END_IF

(*=======================================================*)
	4:	(* Spezifische NC-Achsparameter auslesen *)
		IF fb_state_entry.E THEN
			fb_axis.i16_nc_parameter_nummer := MaxAccelerationSystem;
			st_drive_cmd.enu_cmd := READ_NC_PARAMETER;
		END_IF

		(*-----------------------Weiterschaltbedingungen----------------------------*)
		IF st_drive_cmd.enu_cmd = NO_COMMAND THEN
			st_geschwindigkeiten.lr_beschleunigung := fb_axis.r_wert_nc_read_parameter;
			fb_state_entry.i16_next_step := 5;
		END_IF

(*=======================================================*)
	5:	(* Spezifische NC-Achsparameter auslesen *)
		IF fb_state_entry.E THEN
			fb_axis.i16_nc_parameter_nummer := MaxDecelerationSystem;
			st_drive_cmd.enu_cmd := READ_NC_PARAMETER;
		END_IF

		(*-----------------------Weiterschaltbedingungen----------------------------*)
		IF st_drive_cmd.enu_cmd = NO_COMMAND THEN
			st_geschwindigkeiten.lr_verzoegerung := fb_axis.r_wert_nc_read_parameter;
			lr_decceleration_normal := st_geschwindigkeiten.lr_verzoegerung;
			lr_decceleration_nothalt := 200000.0;
			fb_state_entry.i16_next_step := 6;
		END_IF

(*=======================================================*)
	6:	(* Spezifische NC-Achsparameter auslesen *)
		IF fb_state_entry.E THEN
			fb_axis.i16_nc_parameter_nummer := MaxJerk;
			st_drive_cmd.enu_cmd := READ_NC_PARAMETER;
		END_IF

		(*-----------------------Weiterschaltbedingungen----------------------------*)
		IF st_drive_cmd.enu_cmd = NO_COMMAND THEN
			st_geschwindigkeiten.lr_ruck := fb_axis.r_wert_nc_read_parameter;
			fb_state_entry.i16_next_step := 7;
		END_IF

(*=======================================================*)
	7:	(* Konfigurationen der Achse *)
		IF fb_state_entry.E THEN
			fb_axis.st_eccoe_sdo.s_ec_slave_net_id := ST_EthercatDiag.s_ec_slave_net_id[2];
			fb_axis.st_eccoe_sdo.ui16_slave_addr := st_config_achse.ui16_ethercat_adr;
		END_IF

		(*-----------------------Weiterschaltbedingungen----------------------------*)
		fb_state_entry.i16_next_step := FEHLER; (*in Fehler gehen damit die Achsen resetet werden. Sonst steigen die Achsen bei einem TC Restart aus*)

(*=======================================================*)
	INIT:
		IF fb_state_entry.E THEN
			fb_ton_wz.IN := FALSE;
			fb_ton_uez.IN	:= FALSE;
			fb_ton_quitt.IN := FALSE;
			fb_ton_wz_disable.IN := FALSE;
			st_ctrl_out.b_fehler := FALSE;
			st_ctrl_out.b_fertig := FALSE;
			st_ctrl_out.b_bereit := FALSE;
			st_ctrl_out.b_prebereit := FALSE;

 			fb_axis.lr_soll_geschwindigkeit := gst_datensatz.st_wkz.r_auto;

			st_geschwindigkeiten.lr_verzoegerung := lr_decceleration_normal;

			(* Reset Stoermeldungen *)
			st_sm.b_achse_nicht_auf_startpos := FALSE;
			st_sm.b_achsfehler := FALSE;
			st_sm.b_devicefehler := FALSE;
			st_sm.b_keine_verfahrfreigabe := FALSE;
			st_sm.b_ende_skalierungs_nocke := FALSE;
			st_sm.b_ende_camming_nocke := FALSE;
			st_sm.b_skalierung_noch_aktiv := FALSE;

			sm_fehler_initialposition_achse := FALSE;
			sm_keine_nocken_definiert := FALSE;

		END_IF

		(*-----------------------Weiterschaltbedingungen----------------------------*)
		IF st_ctrl_in.b_preinit THEN
			fb_axis.lr_soll_geschwindigkeit := gst_datensatz.st_wkz.r_auto;
			fb_state_entry.i16_next_step := 15;
		END_IF

(*=======================================================*)
	15:	(* Reglerfreigabe wegnehmen *)
		IF fb_state_entry.E THEN
			st_drive_cmd.enu_cmd := POWER_DISABLE;
		END_IF

		(*-----------------------Weiterschaltbedingungen----------------------------*)
		IF st_drive_cmd.enu_cmd = NO_COMMAND THEN
			fb_state_entry.i16_next_step := 20;
		END_IF

(*=======================================================*)
	20:	(* Überprüfe Nullpunktverschiebung des Absolutwertgebers auf Korrektheit *)
		IF fb_state_entry.E THEN
			fb_axis.i16_nc_parameter_nummer := AxisEncoderOffset;	(* vom Datentyp MC_AxisParameter *)
			st_drive_cmd.enu_cmd := READ_NC_PARAMETER;
		END_IF

		(*-----------------------Weiterschaltbedingungen----------------------------*)
		IF st_drive_cmd.enu_cmd = NO_COMMAND THEN
			IF fb_axis.r_wert_nc_read_parameter = gst_datensatz.st_md.st_md_bestueckachse.lr_nullpunktverschiebung THEN
				fb_state_entry.i16_next_step := 45;	(* Reglerfreigabe setzen *)
			ELSE
				fb_state_entry.i16_next_step := 30;	(* Nullpunktverschiebung schreiben *)
			END_IF
		END_IF
(*
(*=======================================================*)
	25:	(* Überprüfung der Achsposition mit Referenzsensor *)

		(*-----------------------Weiterschaltbedingungen----------------------------*)
		IF e_referenz_sensor THEN
			fb_state_entry.i16_next_step := 30;	(* Achse steht im korrekten Winkelbereich *)
		ELSE
			sm_fehler_initialposition_achse := TRUE;
			fb_state_entry.i16_next_step := FEHLER;	(* Achsposition ist um Vielfache von 72° verschoben *)
		END_IF
*)
(*=======================================================*)
	30:	(* Nullpunktverschiebung hat sich geändert, deshalb erst Null reinschreiben, um keinen Additionsfehler zu machen, *)
		(* weil der Wert der Verschiebung beim Neustart komplett auf die Achse geschrieben wird *)
		IF fb_state_entry.E THEN
			fb_axis.i16_nc_parameter_nummer := AxisEncoderOffset;
			fb_axis.r_wert_nc_write_parameter := 0.0;
			st_drive_cmd.enu_cmd := WRITE_NC_PARAMETER;
		END_IF

		(*-----------------------Weiterschaltbedingungen----------------------------*)
		IF st_drive_cmd.enu_cmd = NO_COMMAND THEN
			fb_state_entry.i16_next_step := 40;
		END_IF

(*=======================================================*)
	40:	(* Aktuelle Nullpunktverschiebung des Absolutwertgebers an die Achse senden *)
		IF fb_state_entry.E THEN
			fb_axis.i16_nc_parameter_nummer := AxisEncoderOffset;
			fb_axis.r_wert_nc_write_parameter := gst_datensatz.st_md.st_md_bestueckachse.lr_nullpunktverschiebung;
			st_drive_cmd.enu_cmd := WRITE_NC_PARAMETER;
		END_IF

		(*-----------------------Weiterschaltbedingungen----------------------------*)
		IF st_drive_cmd.enu_cmd = NO_COMMAND THEN
			fb_state_entry.i16_next_step := 45;
		END_IF

(*=======================================================*)
	45:	(* Reglerfreigabe setzen , Reset wird bei Bedarf automatisch ausgeführt*)
		IF fb_state_entry.E THEN
			st_drive_cmd.enu_cmd := POWER_ENABLE;
		END_IF

		(*-----------------------Weiterschaltbedingungen----------------------------*)
		IF st_drive_cmd.enu_cmd = NO_COMMAND THEN
			fb_state_entry.i16_next_step := 50;
		END_IF

(*=======================================================*)
	50:
		IF fb_state_entry.E THEN
			st_ctrl_out.b_prebereit := TRUE;
		END_IF

		(*-----------------------Weiterschaltbedingungen----------------------------*)
		IF st_ctrl_in.b_init THEN
			fb_state_entry.i16_next_step := 60;
		END_IF

(*=======================================================*)
	60:	(* Überprüfe, ob überhaupt Nocken angelegt sind *)
		IF fb_state_entry.E THEN
			b_nullnockenmerker := TRUE;
			FOR i := 0  TO 5 BY 1DO
				b_nullnockenmerker :=	b_nullnockenmerker AND
								 	gst_datensatz.st_wkz.nockenschaltwerk_bestueckachse.arr_nocken[i].r_cam_begin = 0 AND
									gst_datensatz.st_wkz.nockenschaltwerk_bestueckachse.arr_nocken[i].r_cam_end = 0;
			END_FOR
		END_IF

		(*-----------------------Weiterschaltbedingungen----------------------------*)
		IF b_nullnockenmerker	THEN
			sm_keine_nocken_definiert := TRUE;
			 fb_state_entry.i16_next_step := FEHLER;
		ELSE
			fb_state_entry.i16_next_step := 70;
		END_IF

(*=======================================================*)
	70: (* Alle Nocken einschalten *)
		IF fb_state_entry.E THEN
			FOR i := 0  TO (SIZEOF (nockenschaltwerk_bestueckachse.fb.arr_spur) / SIZEOF (nockenschaltwerk_bestueckachse.fb.arr_spur[0])) - 1 BY 1DO
				gst_datensatz.st_wkz.nockenschaltwerk_bestueckachse.arr_nocken[i].b_camvalid := TRUE;
				gst_datensatz.st_wkz.nockenschaltwerk_bestueckachse.arr_nocken[i].b_eff_direction_neg := TRUE;
				gst_datensatz.st_wkz.nockenschaltwerk_bestueckachse.arr_nocken[i].b_eff_direction_pos := TRUE;
				gst_datensatz.st_wkz.nockenschaltwerk_bestueckachse.arr_nocken[i].i16_track_no := i;
			END_FOR
			(* Nachbearbeitung von bestimmten Nocken *)
			gst_datensatz.st_wkz.nockenschaltwerk_bestueckachse.arr_nocken[NO_OT].b_eff_direction_neg := FALSE;

			(* Zylinder für Bandeinzug mit Vorsteuerzeit belegen *)
			(* 1700 *)
			CASE gst_datensatz.st_wkz.i16_typ_bandeinzug OF
				KEIN_EINZUG:
					;

				STANDARD_2FACH_V2:
					gst_datensatz.st_wkz.nockenschaltwerk_bestueckachse.arr_nocken[NO_BW_BANDFAENGER_LI_BAEZV2_EINFAHREN].t_vorsteuerzeit := t#16ms;
					gst_datensatz.st_wkz.nockenschaltwerk_bestueckachse.arr_nocken[NO_BW_BANDFAENGER_LI_BAEZV2_AUSFAHREN].t_vorsteuerzeit := t#16ms;
					gst_datensatz.st_wkz.nockenschaltwerk_bestueckachse.arr_nocken[NO_BW_BANDKLEMMEN_LI_BAEZV2_EINFAHREN].t_vorsteuerzeit := t#16ms;
					gst_datensatz.st_wkz.nockenschaltwerk_bestueckachse.arr_nocken[NO_BW_BANDKLEMMEN_LI_BAEZV2_AUSFAHREN].t_vorsteuerzeit := t#16ms;
					gst_datensatz.st_wkz.nockenschaltwerk_bestueckachse.arr_nocken[NO_BW_BANDFAENGER_RE_BAEZV2_EINFAHREN].t_vorsteuerzeit := t#16ms;
					gst_datensatz.st_wkz.nockenschaltwerk_bestueckachse.arr_nocken[NO_BW_BANDFAENGER_RE_BAEZV2_AUSFAHREN].t_vorsteuerzeit := t#16ms;
					gst_datensatz.st_wkz.nockenschaltwerk_bestueckachse.arr_nocken[NO_BW_BANDKLEMMEN_RE_BAEZV2_EINFAHREN].t_vorsteuerzeit := t#16ms;
					gst_datensatz.st_wkz.nockenschaltwerk_bestueckachse.arr_nocken[NO_BW_BANDKLEMMEN_RE_BAEZV2_AUSFAHREN].t_vorsteuerzeit := t#16ms;

				BANDWECHSLER_V2:
					(* Bandwechsler V2 ohne Sensoren und anderen Zylindern *)
					gst_datensatz.st_wkz.nockenschaltwerk_bestueckachse.arr_nocken[NO_BW_BANDFAENGER_BAWEV2_EINFAHREN].t_vorsteuerzeit := t#16ms;
					gst_datensatz.st_wkz.nockenschaltwerk_bestueckachse.arr_nocken[NO_BW_BANDFAENGER_BAWEV2_AUSFAHREN].t_vorsteuerzeit := t#16ms;
					gst_datensatz.st_wkz.nockenschaltwerk_bestueckachse.arr_nocken[NO_BW_BANDKLEMMEN_BAWEV2_EINFAHREN].t_vorsteuerzeit := t#16ms;
					gst_datensatz.st_wkz.nockenschaltwerk_bestueckachse.arr_nocken[NO_BW_BANDKLEMMEN_BAWEV2_AUSFAHREN].t_vorsteuerzeit := t#16ms;

				SERVO:
					;
(*					gst_datensatz.st_wkz.nockenschaltwerk_bestueckachse.arr_nocken[NO_SERVOBANDEINZUG_LUEFTEN].r_cam_begin := 135;
					gst_datensatz.st_wkz.nockenschaltwerk_bestueckachse.arr_nocken[NO_SERVOBANDEINZUG_LUEFTEN].r_cam_end := 178;
					gst_datensatz.st_wkz.nockenschaltwerk_bestueckachse.arr_nocken[NO_SERVOBANDEINZUG_GLS].r_cam_begin := 50;
					gst_datensatz.st_wkz.nockenschaltwerk_bestueckachse.arr_nocken[NO_SERVOBANDEINZUG_GLS].r_cam_end := 100;*)
			END_CASE;

			(*-----------------------Weiterschaltbedingungen----------------------------*)
			fb_state_entry.i16_next_step := 80;
		END_IF

(*=======================================================*)
	80:  (* Auf Startposition fahren *)
		CASE gst_datensatz.st_md.i16_typ_zelle OF
			KEINE_ZELLE:
				;

			BESTUECKZELLE_1700, RASTERFOLIE:
				IF fb_state_entry.E THEN
					st_drive_cmd.enu_cmd := MOVE_MODULO;
					fb_axis.mc_richtung_modulo := MC_Shortest_Way ;
					fb_axis.st_position.r_soll := gst_datensatz.st_md.st_md_bestueckachse.lr_startposition;
				END_IF

			BESTUECKZELLE_1720:
				IF fb_state_entry.E THEN
					IF bestueckachse.NcToPlc.ModuloActPos > 0 AND bestueckachse.NcToPlc.ModuloActPos < 90 THEN
						fb_axis.mc_richtung_modulo := MC_Shortest_Way ;
					ELSE
						fb_axis.mc_richtung_modulo := MC_Positive_Direction;
					END_IF
					st_drive_cmd.enu_cmd := MOVE_MODULO;
					fb_axis.st_position.r_soll := gst_datensatz.st_md.st_md_bestueckachse.lr_startposition;
				END_IF
		END_CASE

		(*-----------------------Weiterschaltbedingungen----------------------------*)
		IF st_drive_cmd.enu_cmd = NO_COMMAND THEN
			fb_state_entry.i16_next_step := 90;
		END_IF

(*=======================================================*)
	90:	(* Finale Überprüfung der Achsposition auf Bereich OT oder UT *)

		(*-----------------------Weiterschaltbedingungen----------------------------*)
		IF e_referenz_sensor AND
			bestueckachse.NcToPlc.ModuloActPos >= 0 AND
			bestueckachse.NcToPlc.ModuloActPos < 71.99 THEN
			fb_state_entry.i16_next_step := BEREIT;	(* Achse steht im korrekten Winkelbereich *)
		ELSE
			sm_fehler_initialposition_achse := TRUE;
			fb_state_entry.i16_next_step := FEHLER;	(* Achsposition ist um Vielfache von 72° verschoben *)
		END_IF

(*=======================================================*)
	BEREIT:
		IF fb_state_entry.E THEN
			st_ctrl_out.b_bereit := TRUE;
			st_ctrl_out.b_fertig := TRUE;
		END_IF

(*=======================================================*)
	FEHLER:
		IF fb_state_entry.E THEN
			st_ctrl_out.b_fehler := TRUE;
			fb_ton_quitt.IN := FALSE;
		END_IF

		(*-----------------------Weiterschaltbedingungen----------------------------*)
		IF st_ctrl_in.b_quitt AND NOT fb_state_entry.E THEN
			st_ctrl_out.b_fehler := FALSE;
			st_drive_cmd.enu_cmd := RESET;
			fb_ton_quitt.IN := TRUE;
		END_IF

		IF st_ctrl_in.b_stop AND NOT bestueckachse.Status.HasBeenStopped THEN
			st_drive_cmd.enu_cmd := STOP_AXIS;
		END_IF

		IF st_ctrl_in.b_halt AND bestueckachse.Status.Moving THEN
			st_drive_cmd.enu_cmd := HALT_AXIS;
			st_geschwindigkeiten.lr_verzoegerung := lr_decceleration_nothalt;
		END_IF

		IF fb_ton_quitt.Q THEN
			fb_ton_quitt.IN := FALSE;
			fb_state_entry.i16_next_step := INIT;
		END_IF

(*=======================================================*)
	STOP:
		IF fb_state_entry.E THEN
			IF bestueckachse.NcToPlc.CoupleState = 0 THEN
				st_drive_cmd.enu_cmd := STOP_AXIS;
			END_IF
		END_IF

		(*-----------------------Weiterschaltbedingungen----------------------------*)
		IF st_drive_cmd.enu_cmd = NO_COMMAND AND bestueckachse.Status.NotMoving THEN
			fb_state_entry.i16_next_step := STILLSTAND;
		END_IF

(*=======================================================*)
	STILLSTAND:
		IF fb_state_entry.E THEN
			st_drive_cmd.enu_cmd := POWER_DISABLE;
			fb_ton_quitt.IN := FALSE;
		END_IF

		(*-----------------------Weiterschaltbedingungen----------------------------*)
		IF st_ctrl_in.b_quitt AND NOT fb_state_entry.E THEN
			fb_ton_quitt.IN := TRUE;
		END_IF

		IF fb_ton_quitt.Q THEN
			fb_ton_quitt.IN := FALSE;
			fb_state_entry.i16_next_step := INIT;
		END_IF

(*=======================================================*)
	HALT:
		IF fb_state_entry.E THEN
			IF bestueckachse.NcToPlc.CoupleState = 0 THEN
				st_drive_cmd.enu_cmd := HALT_AXIS;
				st_geschwindigkeiten.lr_verzoegerung := lr_decceleration_nothalt;
			END_IF
			fb_ton_quitt.IN := FALSE;
		END_IF

		(*-----------------------Weiterschaltbedingungen----------------------------*)
		IF st_ctrl_in.b_quitt AND NOT fb_state_entry.E THEN
			fb_ton_quitt.IN := TRUE;
		END_IF

		IF fb_ton_quitt.Q THEN
			fb_ton_quitt.IN := FALSE;
			fb_state_entry.i16_next_step := INIT;
		END_IF

(*=======================================================*)
	HANDRAD:	(* Überprüfe Nullpunktverschiebung des Absolutwertgebers auf Korrektheit *)
		IF fb_state_entry.E THEN
			st_ctrl_out.b_fehler := TRUE;
			fb_axis.i16_nc_parameter_nummer := AxisEncoderOffset;
			st_drive_cmd.enu_cmd := READ_NC_PARAMETER;
		END_IF

		(*-----------------------Weiterschaltbedingungen----------------------------*)
		IF st_drive_cmd.enu_cmd = NO_COMMAND THEN
			IF fb_axis.r_wert_nc_read_parameter = gst_datensatz.st_md.st_md_bestueckachse.lr_nullpunktverschiebung THEN
				fb_state_entry.i16_next_step := 2040;	(* Jogbetrieb *)
			ELSE
				fb_state_entry.i16_next_step := 2010;	(* Reglerfreigabe nehmen und Nullpunktverschiebung schreiben *)
			END_IF
		END_IF

(*=======================================================*)
	2010:	(* Reglerfreigabe wegnehmen , damit Nullpunktverschiebung geschrieben werden kannt*)
		IF fb_state_entry.E THEN
			st_drive_cmd.enu_cmd := POWER_DISABLE;
		END_IF

		(*-----------------------Weiterschaltbedingungen----------------------------*)
		IF st_drive_cmd.enu_cmd = NO_COMMAND THEN
			fb_state_entry.i16_next_step := 2020;
		END_IF

(*=======================================================*)
	2020:	(* Nullpunktverschiebung hat sich geändert, deshalb erst Null reinschreiben, um keinen Additionsfehler zu machen, *)
			(* weil der Wert der Verschiebung beim Neustart komplett auf die Achse geschrieben wird *)
		IF fb_state_entry.E THEN
			fb_axis.i16_nc_parameter_nummer := AxisEncoderOffset;
			fb_axis.r_wert_nc_write_parameter := 0.0;
			st_drive_cmd.enu_cmd := WRITE_NC_PARAMETER;
		END_IF

		(*-----------------------Weiterschaltbedingungen----------------------------*)
		IF st_drive_cmd.enu_cmd = NO_COMMAND THEN
			fb_state_entry.i16_next_step := 2030;
		END_IF

(*=======================================================*)
	2030:	(* Aktuelle Nullpunktverschiebung des Absolutwertgebers an die Achse senden *)
		IF fb_state_entry.E THEN
			fb_axis.i16_nc_parameter_nummer := AxisEncoderOffset;
			fb_axis.r_wert_nc_write_parameter := gst_datensatz.st_md.st_md_bestueckachse.lr_nullpunktverschiebung;
			st_drive_cmd.enu_cmd := WRITE_NC_PARAMETER;
		END_IF

		(*-----------------------Weiterschaltbedingungen----------------------------*)
		IF st_drive_cmd.enu_cmd = NO_COMMAND THEN
			fb_state_entry.i16_next_step := 2040;
		END_IF

(*=======================================================*)
	2040:	(* Jogbetrieb *)
		IF fb_state_entry.E THEN
			fb_axis.lr_soll_geschwindigkeit := st_geschwindigkeiten.lr_jog;
		END_IF

		IF ST_Euchner_Handbedienpult.i16_Handrad_delta > 0 THEN
			st_drive_cmd.enu_cmd := JOG_VORWAERTS;
		ELSIF ST_Euchner_Handbedienpult.i16_Handrad_delta < 0 THEN
			st_drive_cmd.enu_cmd := JOG_RUECKWAERTS;
		ELSE
			IF bestueckachse.Status.Moving THEN
				st_drive_cmd.enu_cmd := JOG_STOP;
			END_IF
		END_IF

		IF fb_r_trig_taste_plus.Q THEN
			fb_state_entry.i16_next_step := MOTORBREMSE_AUF;
		END_IF
		IF fb_r_trig_taste_minus.Q THEN
			fb_state_entry.i16_next_step := MOTORBREMSE_ZU;
		END_IF

		(*-----------------------Weiterschaltbedingungen----------------------------*)
		IF gi16_betriebsart <> HAND OR NOT b_hand_dialog_aktiv THEN
			fb_state_entry.i16_next_step := 2050;
		END_IF

(*=======================================================*)
	2050:
		IF fb_state_entry.E THEN
			st_drive_cmd.enu_cmd := ABORT;
		END_IF

		(*-----------------------Weiterschaltbedingungen----------------------------*)
		IF st_drive_cmd.enu_cmd = NO_COMMAND THEN
			fb_state_entry.i16_next_step := 2060;
		END_IF

(*=======================================================*)
	2060:
		IF fb_state_entry.E THEN
			fb_axis.w_idn := P_0_IDN + 96;
			fb_axis.ui16_soeparam_write_value := 0;	(* Motorbremse im Automatikbetrieb für reguläres Fahren *)
			st_drive_cmd.enu_cmd := SOE_WRITE_PARAM;
		END_IF

		(*-----------------------Weiterschaltbedingungen----------------------------*)
		IF st_drive_cmd.enu_cmd = NO_COMMAND THEN
			fb_state_entry.i16_next_step := 2070;
		END_IF

(*=======================================================*)
	2070:	(* Reglerfreigabe wegnehmen *)
		IF fb_state_entry.E THEN
			st_drive_cmd.enu_cmd := POWER_DISABLE;
		END_IF

		(*-----------------------Weiterschaltbedingungen----------------------------*)
		IF st_drive_cmd.enu_cmd = NO_COMMAND THEN
			st_ctrl_out.b_fehler := FALSE;
			fb_state_entry.i16_next_step := INIT;
		END_IF

(*=======================================================*)
	MOTORBREMSE_AUF:
		IF fb_state_entry.E THEN
			st_drive_cmd.enu_cmd := ABORT;
		END_IF

		(*-----------------------Weiterschaltbedingungen----------------------------*)
		IF st_drive_cmd.enu_cmd = NO_COMMAND THEN
			fb_state_entry.i16_next_step := 2110;
		END_IF

(*=======================================================*)
	2110:	(* Reglerfreigabe wegnehmen *)
		IF fb_state_entry.E THEN
			st_drive_cmd.enu_cmd := POWER_DISABLE;
		END_IF

		(*-----------------------Weiterschaltbedingungen----------------------------*)
		IF st_drive_cmd.enu_cmd = NO_COMMAND THEN
			fb_state_entry.i16_next_step := 2120;
		END_IF

(*=======================================================*)
	2120:	(* Bremse auf machen *)
		IF fb_state_entry.E THEN
			fb_axis.w_idn := P_0_IDN + 96;
			fb_axis.ui16_soeparam_write_value := 2;
			st_drive_cmd.enu_cmd := SOE_WRITE_PARAM;
		END_IF

		(*-----------------------Weiterschaltbedingungen----------------------------*)
		IF 	st_drive_cmd.enu_cmd = NO_COMMAND AND
			(gi16_betriebsart <> HAND OR
			NOT b_hand_dialog_aktiv OR
			ST_Euchner_Handbedienpult.i16_Handrad_delta > 0)
			THEN
				fb_state_entry.i16_next_step := HANDRAD;
		ELSIF fb_r_trig_taste_minus.Q THEN
			fb_state_entry.i16_next_step := MOTORBREMSE_ZU;
		END_IF

(*=======================================================*)
	MOTORBREMSE_ZU:
		IF fb_state_entry.E THEN
			st_drive_cmd.enu_cmd := ABORT;
		END_IF

		(*-----------------------Weiterschaltbedingungen----------------------------*)
		IF st_drive_cmd.enu_cmd = NO_COMMAND THEN
			fb_state_entry.i16_next_step := 2210;
		END_IF

(*=======================================================*)
	2210:	(* Reglerfreigabe setzen *)
		IF fb_state_entry.E THEN
			st_drive_cmd.enu_cmd := POWER_ENABLE;
		END_IF

		(*-----------------------Weiterschaltbedingungen----------------------------*)
		IF st_drive_cmd.enu_cmd = NO_COMMAND THEN
			fb_state_entry.i16_next_step := 2220;
		END_IF

(*=======================================================*)
	2220:	(* Bremse zu machen *)
		IF fb_state_entry.E THEN
			fb_axis.w_idn := P_0_IDN + 96;
			fb_axis.ui16_soeparam_write_value := 0;	(* Motorbremse im Automatikbetrieb für reguläres Fahren *)
			st_drive_cmd.enu_cmd := SOE_WRITE_PARAM;
		END_IF

		(*-----------------------Weiterschaltbedingungen----------------------------*)
		IF 	st_drive_cmd.enu_cmd = NO_COMMAND AND
			(gi16_betriebsart <> HAND OR
			NOT b_hand_dialog_aktiv OR
			ST_Euchner_Handbedienpult.i16_Handrad_delta > 0)
			THEN
				fb_state_entry.i16_next_step := HANDRAD;
		ELSIF fb_r_trig_taste_plus.Q THEN
			fb_state_entry.i16_next_step := MOTORBREMSE_AUF;
		END_IF

(*=======================================================*)
	NULLPUNKT_SETZEN:
		(* Aktuellen Jog beenden, sonst Probleme beim Softwareendschalter*)
		IF fb_state_entry.E THEN
			st_drive_cmd.enu_cmd := JOG_STOP;
		END_IF

		(*-----------------------Weiterschaltbedingungen----------------------------*)
		IF st_drive_cmd.enu_cmd = NO_COMMAND THEN
			fb_state_entry.i16_next_step := 2505;
		END_IF

(*=======================================================*)
	2505:
		(* 	Lese aktuelle Nullpunkt verschiebung von der Hardware. Der Benutze könnte einen falschen
			Wert eingetragen haben *)
		IF fb_state_entry.E THEN
			fb_axis.i16_nc_parameter_nummer := AxisEncoderOffset;
			st_drive_cmd.enu_cmd := READ_NC_PARAMETER;
		END_IF

		(*-----------------------Weiterschaltbedingungen----------------------------*)
		IF st_drive_cmd.enu_cmd = NO_COMMAND THEN
			gst_datensatz.st_md.st_md_bestueckachse.lr_nullpunktverschiebung := fb_axis.r_wert_nc_read_parameter;
			fb_state_entry.i16_next_step := 2510;
		END_IF

(*=======================================================*)
	2510:	(* Nullpunktverschiebung berechnen *)
		IF fb_state_entry.E THEN
			lr_pos_ohneverschiebung := axis_bestueckachse.st_visu.lr_position_ist - gst_datensatz.st_md.st_md_bestueckachse.lr_nullpunktverschiebung;
		
			gst_datensatz.st_md.st_md_bestueckachse.lr_nullpunktverschiebung := - lr_pos_ohneverschiebung;
	
			WHILE (gst_datensatz.st_md.st_md_bestueckachse.lr_nullpunktverschiebung > 360)
			DO
				gst_datensatz.st_md.st_md_bestueckachse.lr_nullpunktverschiebung :=
					gst_datensatz.st_md.st_md_bestueckachse.lr_nullpunktverschiebung - 360;
			END_WHILE
		
			WHILE (gst_datensatz.st_md.st_md_bestueckachse.lr_nullpunktverschiebung < 0)
			DO
				gst_datensatz.st_md.st_md_bestueckachse.lr_nullpunktverschiebung :=
					gst_datensatz.st_md.st_md_bestueckachse.lr_nullpunktverschiebung + 360;
			END_WHILE
		END_IF

		(*-----------------------Weiterschaltbedingungen----------------------------*)
		(* Aktiviere den wert in die Hardware *)
		fb_state_entry.i16_next_step := HANDRAD;

(*=======================================================*)
	INBETRIEBNAHME:	(* Überprüfe Nullpunktverschiebung des Absolutwertgebers auf Korrektheit *)
		IF fb_state_entry.E THEN
			fb_axis.i16_nc_parameter_nummer := AxisEncoderOffset;
			st_drive_cmd.enu_cmd := READ_NC_PARAMETER;
		END_IF

		(*-----------------------Weiterschaltbedingungen----------------------------*)
		IF st_drive_cmd.enu_cmd = NO_COMMAND THEN
			IF fb_axis.r_wert_nc_read_parameter = gst_datensatz.st_md.st_md_bestueckachse.lr_nullpunktverschiebung THEN
				fb_state_entry.i16_next_step := 5100;	(* Reversiersequenz*)
			ELSE
				fb_state_entry.i16_next_step := 5010;	(* Reglerfreigabe nehmen und Nullpunktverschiebung schreiben *)
			END_IF
		END_IF

(*=======================================================*)
	5010:	(* Reglerfreigabe wegnehmen, damit Nullpunktverschiebung geschrieben werden kannt*)
		IF fb_state_entry.E THEN
			st_drive_cmd.enu_cmd := POWER_DISABLE;
		END_IF

		(*-----------------------Weiterschaltbedingungen----------------------------*)
		IF st_drive_cmd.enu_cmd = NO_COMMAND THEN
			fb_state_entry.i16_next_step := 5020;
		END_IF

(*=======================================================*)
	5020:	(* Nullpunktverschiebung hat sich geändert, deshalb erst Null reinschreiben, um keinen Additionsfehler zu machen, *)
			(* weil der Wert der Verschiebung beim Neustart komplett auf die Achse geschrieben wird *)
		IF fb_state_entry.E THEN
			fb_axis.i16_nc_parameter_nummer := AxisEncoderOffset;
			fb_axis.r_wert_nc_write_parameter := 0.0;
			st_drive_cmd.enu_cmd := WRITE_NC_PARAMETER;
		END_IF

		(*-----------------------Weiterschaltbedingungen----------------------------*)
		IF st_drive_cmd.enu_cmd = NO_COMMAND THEN
			fb_state_entry.i16_next_step := 5030;
		END_IF

(*=======================================================*)
	5030:	(* Aktuelle Nullpunktverschiebung des Absolutwertgebers an die Achse senden *)
		IF fb_state_entry.E THEN
			fb_axis.i16_nc_parameter_nummer := AxisEncoderOffset;
			fb_axis.r_wert_nc_write_parameter := gst_datensatz.st_md.st_md_bestueckachse.lr_nullpunktverschiebung;
			st_drive_cmd.enu_cmd := WRITE_NC_PARAMETER;
		END_IF

		(*-----------------------Weiterschaltbedingungen----------------------------*)
		IF st_drive_cmd.enu_cmd = NO_COMMAND THEN
			fb_state_entry.i16_next_step := 5100;
		END_IF

(*=======================================================*)
	5100:	(* Verfahren der Achse zwischen zwei Punkten zum Testen verschiedener Achsparameter *)
		IF fb_state_entry.E THEN
			fb_axis.lr_soll_geschwindigkeit := st_geschwindigkeiten.lr_jog;
			fb_axis.st_position.lr_ibn_pos_start := 0.0;
			fb_axis.st_position.lr_ibn_pos_ziel := 180.0;
		END_IF

		(*-----------------------Weiterschaltbedingungen----------------------------*)
		IF st_ctrl_in.b_ibn_start THEN
			fb_state_entry.i16_next_step := 5110;
		END_IF

(*=======================================================*)
	5110: (* Fahre Bestückachse auf Startposition *)
(*
		IF fb_state_entry.E THEN
			 fb_axis.st_position.r_soll := fb_axis.st_position.lr_ibn_pos_start;
			fb_axis.mc_richtung_modulo :=MC_Positive_Direction ;
			st_drive_cmd.enu_cmd := MOVE_MODULO;
		END_IF

		(*-----------------------Weiterschaltbedingungen----------------------------*)
		IF st_drive_cmd.enu_cmd = NO_COMMAND THEN
			fb_state_entry.i16_next_step := 5120;
		END_IF
*)
		IF fb_state_entry.E THEN
			st_drive_cmd.enu_cmd := POWER_ENABLE;
		END_IF

		(*-----------------------Weiterschaltbedingungen----------------------------*)
		IF st_drive_cmd.enu_cmd = NO_COMMAND THEN
			;
		END_IF

(*=======================================================*)
	5120: (* Pause *)
		IF fb_state_entry.E THEN
			fb_ton_wz.PT := t#1s;
			fb_ton_wz.IN := TRUE;
		END_IF

		(*-----------------------Weiterschaltbedingungen----------------------------*)
		IF fb_ton_wz.Q THEN
			fb_ton_wz.IN := FALSE;
			fb_state_entry.i16_next_step := 5130;
		END_IF

(*=======================================================*)
	5130: (* Fahre Bestückachse auf Zielposition *)
		IF fb_state_entry.E THEN
			 fb_axis.st_position.r_soll := fb_axis.st_position.lr_ibn_pos_ziel;
			fb_axis.mc_richtung_modulo :=MC_Negative_Direction ;
			st_drive_cmd.enu_cmd := MOVE_MODULO;
		END_IF

		(*-----------------------Weiterschaltbedingungen----------------------------*)
		IF st_drive_cmd.enu_cmd = NO_COMMAND THEN
			fb_state_entry.i16_next_step := 5140;
		END_IF

(*=======================================================*)
	5140: (* Pause *)
		IF fb_state_entry.E THEN
			fb_ton_wz.PT := t#1s;
			fb_ton_wz.IN := TRUE;
		END_IF

		(*-----------------------Weiterschaltbedingungen----------------------------*)
		IF fb_ton_wz.Q THEN
			fb_ton_wz.IN := FALSE;
			fb_state_entry.i16_next_step := 5100;
		END_IF
END_CASE

fb_state_entry(
	i16_next_step:= , 
	i16_pos:= 2,
	s_debugtext:= ,
	E=> ,
	X=> ,
	i16_step=> ,
	i16_last_step=> );

IF st_config_achse.b_config_fertig THEN
	(* Fehlermeldungen und Betriebsmeldungen ab dem Startindex in die globalen Meldungsarrays schreiben *)
	garr_stoermeldungen[st_config_achse.i16_meld_startindex + 0] := st_sm.b_achse_nicht_bb;
	garr_stoermeldungen[st_config_achse.i16_meld_startindex + 1] := st_sm.b_achse_nicht_referenziert;
	garr_stoermeldungen[st_config_achse.i16_meld_startindex + 2] := st_sm.b_keine_verfahrfreigabe;
	garr_stoermeldungen[st_config_achse.i16_meld_startindex + 3] := st_sm.b_achse_nicht_auf_startpos;
	garr_stoermeldungen[st_config_achse.i16_meld_startindex + 4] := st_sm.b_ende_skalierungs_nocke;
	garr_stoermeldungen[st_config_achse.i16_meld_startindex + 5] := st_sm.b_ende_camming_nocke;
	garr_stoermeldungen[st_config_achse.i16_meld_startindex + 6] := st_sm.b_skalierung_noch_aktiv;
	garr_stoermeldungen[st_config_achse.i16_meld_startindex + 7] := FALSE;
	garr_stoermeldungen[st_config_achse.i16_meld_startindex + 8] := FALSE;
	garr_stoermeldungen[st_config_achse.i16_meld_startindex + 9] := FALSE;
	garr_stoermeldungen[st_config_achse.i16_meld_startindex + 10] := FALSE;
	garr_stoermeldungen[st_config_achse.i16_meld_startindex + 11] := FALSE;
	garr_stoermeldungen[st_config_achse.i16_meld_startindex + 12] := sm_fehler_initialposition_achse;
	garr_stoermeldungen[st_config_achse.i16_meld_startindex + 13] := sm_keine_nocken_definiert;
	garr_stoermeldungen[st_config_achse.i16_meld_startindex + 14] := FALSE;
	garr_stoermeldungen[st_config_achse.i16_meld_startindex + 15] := sm_fehler_ot_ut;
	garr_stoermeldungen[st_config_achse.i16_meld_startindex + 16] := st_drive_cmd.meldungen.sm_write_soe_parameter;
	garr_stoermeldungen[st_config_achse.i16_meld_startindex + 17] := st_drive_cmd.meldungen.sm_read_soe_parameter;
	garr_stoermeldungen[st_config_achse.i16_meld_startindex + 18] := st_drive_cmd.meldungen.sm_write_nc_parameter;
	garr_stoermeldungen[st_config_achse.i16_meld_startindex + 19] := st_drive_cmd.meldungen.sm_read_nc_parameter;
	garr_stoermeldungen[st_config_achse.i16_meld_startindex + 20] := st_drive_cmd.meldungen.sm_power_enable;
	garr_stoermeldungen[st_config_achse.i16_meld_startindex + 21] := st_drive_cmd.meldungen.sm_power_disable;
	garr_stoermeldungen[st_config_achse.i16_meld_startindex + 22] := st_drive_cmd.meldungen.sm_reset;
	garr_stoermeldungen[st_config_achse.i16_meld_startindex + 23] := st_drive_cmd.meldungen.sm_home;
	garr_stoermeldungen[st_config_achse.i16_meld_startindex + 24] := st_drive_cmd.meldungen.sm_setposition;
	garr_stoermeldungen[st_config_achse.i16_meld_startindex + 25] := st_drive_cmd.meldungen.sm_jog_vorwaerts;
	garr_stoermeldungen[st_config_achse.i16_meld_startindex + 26] := st_drive_cmd.meldungen.sm_jog_rueckwaerts;
	garr_stoermeldungen[st_config_achse.i16_meld_startindex + 27] := st_drive_cmd.meldungen.sm_move_absolute;
	garr_stoermeldungen[st_config_achse.i16_meld_startindex + 28] := st_drive_cmd.meldungen.sm_move_relative;
	garr_stoermeldungen[st_config_achse.i16_meld_startindex + 29] := st_drive_cmd.meldungen.sm_move_velocity;
	garr_stoermeldungen[st_config_achse.i16_meld_startindex + 30] := st_drive_cmd.meldungen.sm_move_modulo;
	garr_stoermeldungen[st_config_achse.i16_meld_startindex + 31] := st_drive_cmd.meldungen.sm_stop_axis;
	garr_stoermeldungen[st_config_achse.i16_meld_startindex + 32] := st_drive_cmd.meldungen.sm_halt_axis;
	garr_stoermeldungen[st_config_achse.i16_meld_startindex + 33] := st_drive_cmd.meldungen.sm_motion_command_timeout;
	garr_stoermeldungen[st_config_achse.i16_meld_startindex + 34] := st_sm.b_achsfehler;
	garr_stoermeldungen[st_config_achse.i16_meld_startindex + 35] := st_sm.b_devicefehler;
	garr_stoermeldungen[st_config_achse.i16_meld_startindex + 36] := st_drive_cmd.meldungen.sm_limit_positiv_erreicht;
	garr_stoermeldungen[st_config_achse.i16_meld_startindex + 37] := st_drive_cmd.meldungen.sm_limit_negativ_erreicht;
	garr_stoermeldungen[st_config_achse.i16_meld_startindex + 38] := st_drive_cmd.meldungen.sm_ec_coe_sdo_write_ex;
	garr_stoermeldungen[st_config_achse.i16_meld_startindex + 39] := st_drive_cmd.meldungen.sm_ec_coe_sdo_read_ex;
	garr_stoermeldungen[st_config_achse.i16_meld_startindex + 40] := FALSE;
	garr_stoermeldungen[st_config_achse.i16_meld_startindex + 41] := FALSE;
	garr_stoermeldungen[st_config_achse.i16_meld_startindex + 42] := FALSE;
	garr_stoermeldungen[st_config_achse.i16_meld_startindex + 43] := FALSE;
	garr_stoermeldungen[st_config_achse.i16_meld_startindex + 44] := FALSE;
	garr_stoermeldungen[st_config_achse.i16_meld_startindex + 45] := FALSE;
	garr_stoermeldungen[st_config_achse.i16_meld_startindex + 46] := FALSE;
	garr_stoermeldungen[st_config_achse.i16_meld_startindex + 47] := FALSE;
	garr_stoermeldungen[st_config_achse.i16_meld_startindex + 48] := FALSE;
	garr_stoermeldungen[st_config_achse.i16_meld_startindex + 49] := FALSE;
	garr_stoermeldungen[st_config_achse.i16_meld_startindex + 50] := FALSE;
	garr_stoermeldungen[st_config_achse.i16_meld_startindex + 51] := FALSE;
	garr_stoermeldungen[st_config_achse.i16_meld_startindex + 52] := FALSE;
	garr_stoermeldungen[st_config_achse.i16_meld_startindex + 53] := FALSE;
	garr_stoermeldungen[st_config_achse.i16_meld_startindex + 54] := FALSE;
	garr_stoermeldungen[st_config_achse.i16_meld_startindex + 55] := FALSE;
	garr_stoermeldungen[st_config_achse.i16_meld_startindex + 56] := FALSE;
	garr_stoermeldungen[st_config_achse.i16_meld_startindex + 57] := FALSE;
	garr_stoermeldungen[st_config_achse.i16_meld_startindex + 58] := FALSE;
	garr_stoermeldungen[st_config_achse.i16_meld_startindex + 59] := FALSE;
	garr_stoermeldungen[st_config_achse.i16_meld_startindex + 60] := FALSE;
	garr_stoermeldungen[st_config_achse.i16_meld_startindex + 61] := FALSE;
	garr_stoermeldungen[st_config_achse.i16_meld_startindex + 62] := FALSE;
	garr_stoermeldungen[st_config_achse.i16_meld_startindex + 63] := FALSE;
	garr_stoermeldungen[st_config_achse.i16_meld_startindex + 64] := FALSE;
	garr_stoermeldungen[st_config_achse.i16_meld_startindex + 65] := FALSE;
	garr_stoermeldungen[st_config_achse.i16_meld_startindex + 66] := FALSE;
	garr_stoermeldungen[st_config_achse.i16_meld_startindex + 67] := FALSE;
	garr_stoermeldungen[st_config_achse.i16_meld_startindex + 68] := FALSE;
	garr_stoermeldungen[st_config_achse.i16_meld_startindex + 69] := FALSE;
	garr_stoermeldungen[st_config_achse.i16_meld_startindex + 70] :=  FALSE;
	garr_stoermeldungen[st_config_achse.i16_meld_startindex + 71] :=  FALSE;
	garr_stoermeldungen[st_config_achse.i16_meld_startindex + 72] :=  FALSE;
	garr_stoermeldungen[st_config_achse.i16_meld_startindex + 73] :=  FALSE;
	garr_stoermeldungen[st_config_achse.i16_meld_startindex + 74] :=  FALSE;
	garr_stoermeldungen[st_config_achse.i16_meld_startindex + 75] :=  FALSE;
	garr_stoermeldungen[st_config_achse.i16_meld_startindex + 76] :=  FALSE;
	garr_stoermeldungen[st_config_achse.i16_meld_startindex + 77] :=  FALSE;
	garr_stoermeldungen[st_config_achse.i16_meld_startindex + 78] :=  FALSE;
	garr_stoermeldungen[st_config_achse.i16_meld_startindex + 79] :=  FALSE;
	garr_stoermeldungen[st_config_achse.i16_meld_startindex + 80] :=  FALSE;
	garr_stoermeldungen[st_config_achse.i16_meld_startindex + 81] :=  FALSE;
	garr_stoermeldungen[st_config_achse.i16_meld_startindex + 82] :=  FALSE;
	garr_stoermeldungen[st_config_achse.i16_meld_startindex + 83] :=  FALSE;
	garr_stoermeldungen[st_config_achse.i16_meld_startindex + 84] :=  FALSE;
	garr_stoermeldungen[st_config_achse.i16_meld_startindex + 85] :=  FALSE;
	garr_stoermeldungen[st_config_achse.i16_meld_startindex + 86] :=  FALSE;
	garr_stoermeldungen[st_config_achse.i16_meld_startindex + 87] :=  FALSE;
	garr_stoermeldungen[st_config_achse.i16_meld_startindex + 88] :=  FALSE;
	garr_stoermeldungen[st_config_achse.i16_meld_startindex + 89] :=  FALSE;
	garr_stoermeldungen[st_config_achse.i16_meld_startindex + 90] :=  FALSE;
	garr_stoermeldungen[st_config_achse.i16_meld_startindex + 91] :=  FALSE;
	garr_stoermeldungen[st_config_achse.i16_meld_startindex + 92] :=  FALSE;
	garr_stoermeldungen[st_config_achse.i16_meld_startindex + 93] :=  FALSE;
	garr_stoermeldungen[st_config_achse.i16_meld_startindex + 94] :=  FALSE;
	garr_stoermeldungen[st_config_achse.i16_meld_startindex + 95] :=  FALSE;
	garr_stoermeldungen[st_config_achse.i16_meld_startindex + 96] :=  FALSE;
	garr_stoermeldungen[st_config_achse.i16_meld_startindex + 97] :=  FALSE;
	garr_stoermeldungen[st_config_achse.i16_meld_startindex + 98] :=  FALSE;
	garr_stoermeldungen[st_config_achse.i16_meld_startindex + 99] :=  FALSE;

	garr_betriebsmeldungen[st_config_achse.i16_meld_startindex + 0] := FALSE;
	garr_betriebsmeldungen[st_config_achse.i16_meld_startindex + 1] := FALSE;
	garr_betriebsmeldungen[st_config_achse.i16_meld_startindex + 2] := FALSE;
	garr_betriebsmeldungen[st_config_achse.i16_meld_startindex + 3] := FALSE;
	garr_betriebsmeldungen[st_config_achse.i16_meld_startindex + 4] := FALSE;
	garr_betriebsmeldungen[st_config_achse.i16_meld_startindex + 5] := FALSE;
	garr_betriebsmeldungen[st_config_achse.i16_meld_startindex + 6] := FALSE;
	garr_betriebsmeldungen[st_config_achse.i16_meld_startindex + 7] := FALSE;
	garr_betriebsmeldungen[st_config_achse.i16_meld_startindex + 8] := FALSE;
	garr_betriebsmeldungen[st_config_achse.i16_meld_startindex + 9] := FALSE;
	garr_betriebsmeldungen[st_config_achse.i16_meld_startindex + 10] := FALSE;
	garr_betriebsmeldungen[st_config_achse.i16_meld_startindex + 11] := FALSE;
	garr_betriebsmeldungen[st_config_achse.i16_meld_startindex + 12] := FALSE;
	garr_betriebsmeldungen[st_config_achse.i16_meld_startindex + 13] := FALSE;
	garr_betriebsmeldungen[st_config_achse.i16_meld_startindex + 14] := FALSE;
	garr_betriebsmeldungen[st_config_achse.i16_meld_startindex + 15] := FALSE;
	garr_betriebsmeldungen[st_config_achse.i16_meld_startindex + 16] := FALSE;
	garr_betriebsmeldungen[st_config_achse.i16_meld_startindex + 17] := FALSE;
	garr_betriebsmeldungen[st_config_achse.i16_meld_startindex + 18] := FALSE;
	garr_betriebsmeldungen[st_config_achse.i16_meld_startindex + 19] := FALSE;
	garr_betriebsmeldungen[st_config_achse.i16_meld_startindex + 20] := FALSE;
	garr_betriebsmeldungen[st_config_achse.i16_meld_startindex + 21] := FALSE;
	garr_betriebsmeldungen[st_config_achse.i16_meld_startindex + 22] := FALSE;
	garr_betriebsmeldungen[st_config_achse.i16_meld_startindex + 23] := FALSE;
	garr_betriebsmeldungen[st_config_achse.i16_meld_startindex + 24] := FALSE;
	garr_betriebsmeldungen[st_config_achse.i16_meld_startindex + 25] := FALSE;
	garr_betriebsmeldungen[st_config_achse.i16_meld_startindex + 26] := FALSE;
	garr_betriebsmeldungen[st_config_achse.i16_meld_startindex + 27] := FALSE;
	garr_betriebsmeldungen[st_config_achse.i16_meld_startindex + 28] := FALSE;
	garr_betriebsmeldungen[st_config_achse.i16_meld_startindex + 29] := FALSE;
	garr_betriebsmeldungen[st_config_achse.i16_meld_startindex + 30] := FALSE;
	garr_betriebsmeldungen[st_config_achse.i16_meld_startindex + 31] := FALSE;
	garr_betriebsmeldungen[st_config_achse.i16_meld_startindex + 32] := FALSE;
	garr_betriebsmeldungen[st_config_achse.i16_meld_startindex + 33] := FALSE;
	garr_betriebsmeldungen[st_config_achse.i16_meld_startindex + 34] := FALSE;
	garr_betriebsmeldungen[st_config_achse.i16_meld_startindex + 35] := FALSE;
	garr_betriebsmeldungen[st_config_achse.i16_meld_startindex + 36] := FALSE;
	garr_betriebsmeldungen[st_config_achse.i16_meld_startindex + 37] := FALSE;
	garr_betriebsmeldungen[st_config_achse.i16_meld_startindex + 38] := FALSE;
	garr_betriebsmeldungen[st_config_achse.i16_meld_startindex + 39] := FALSE;
	garr_betriebsmeldungen[st_config_achse.i16_meld_startindex + 40] := FALSE;
	garr_betriebsmeldungen[st_config_achse.i16_meld_startindex + 41] := FALSE;
	garr_betriebsmeldungen[st_config_achse.i16_meld_startindex + 42] := FALSE;
	garr_betriebsmeldungen[st_config_achse.i16_meld_startindex + 43] := FALSE;
	garr_betriebsmeldungen[st_config_achse.i16_meld_startindex + 44] := FALSE;
	garr_betriebsmeldungen[st_config_achse.i16_meld_startindex + 45] := FALSE;
	garr_betriebsmeldungen[st_config_achse.i16_meld_startindex + 46] := FALSE;
	garr_betriebsmeldungen[st_config_achse.i16_meld_startindex + 47] := FALSE;
	garr_betriebsmeldungen[st_config_achse.i16_meld_startindex + 48] := FALSE;
	garr_betriebsmeldungen[st_config_achse.i16_meld_startindex + 49] := FALSE;
	garr_betriebsmeldungen[st_config_achse.i16_meld_startindex + 50] := FALSE;
	garr_betriebsmeldungen[st_config_achse.i16_meld_startindex + 51] := FALSE;
	garr_betriebsmeldungen[st_config_achse.i16_meld_startindex + 52] := FALSE;
	garr_betriebsmeldungen[st_config_achse.i16_meld_startindex + 53] := FALSE;
	garr_betriebsmeldungen[st_config_achse.i16_meld_startindex + 54] := FALSE;
	garr_betriebsmeldungen[st_config_achse.i16_meld_startindex + 55] := FALSE;
	garr_betriebsmeldungen[st_config_achse.i16_meld_startindex + 56] := FALSE;
	garr_betriebsmeldungen[st_config_achse.i16_meld_startindex + 57] := FALSE;
	garr_betriebsmeldungen[st_config_achse.i16_meld_startindex + 58] := FALSE;
	garr_betriebsmeldungen[st_config_achse.i16_meld_startindex + 59] := FALSE;
	garr_betriebsmeldungen[st_config_achse.i16_meld_startindex + 60] := FALSE;
	garr_betriebsmeldungen[st_config_achse.i16_meld_startindex + 61] := FALSE;
	garr_betriebsmeldungen[st_config_achse.i16_meld_startindex + 62] := FALSE;
	garr_betriebsmeldungen[st_config_achse.i16_meld_startindex + 63] := FALSE;
	garr_betriebsmeldungen[st_config_achse.i16_meld_startindex + 64] := FALSE;
	garr_betriebsmeldungen[st_config_achse.i16_meld_startindex + 65] := FALSE;
	garr_betriebsmeldungen[st_config_achse.i16_meld_startindex + 66] := FALSE;
	garr_betriebsmeldungen[st_config_achse.i16_meld_startindex + 67] := FALSE;
	garr_betriebsmeldungen[st_config_achse.i16_meld_startindex + 68] := FALSE;
	garr_betriebsmeldungen[st_config_achse.i16_meld_startindex + 69] := FALSE;
	garr_betriebsmeldungen[st_config_achse.i16_meld_startindex + 70] :=  FALSE;
	garr_betriebsmeldungen[st_config_achse.i16_meld_startindex + 71] :=  FALSE;
	garr_betriebsmeldungen[st_config_achse.i16_meld_startindex + 72] :=  FALSE;
	garr_betriebsmeldungen[st_config_achse.i16_meld_startindex + 73] :=  FALSE;
	garr_betriebsmeldungen[st_config_achse.i16_meld_startindex + 74] :=  FALSE;
	garr_betriebsmeldungen[st_config_achse.i16_meld_startindex + 75] :=  FALSE;
	garr_betriebsmeldungen[st_config_achse.i16_meld_startindex + 76] :=  FALSE;
	garr_betriebsmeldungen[st_config_achse.i16_meld_startindex + 77] :=  FALSE;
	garr_betriebsmeldungen[st_config_achse.i16_meld_startindex + 78] :=  FALSE;
	garr_betriebsmeldungen[st_config_achse.i16_meld_startindex + 79] :=  FALSE;
	garr_betriebsmeldungen[st_config_achse.i16_meld_startindex + 80] :=  FALSE;
	garr_betriebsmeldungen[st_config_achse.i16_meld_startindex + 81] :=  FALSE;
	garr_betriebsmeldungen[st_config_achse.i16_meld_startindex + 82] :=  FALSE;
	garr_betriebsmeldungen[st_config_achse.i16_meld_startindex + 83] :=  FALSE;
	garr_betriebsmeldungen[st_config_achse.i16_meld_startindex + 84] :=  FALSE;
	garr_betriebsmeldungen[st_config_achse.i16_meld_startindex + 85] :=  FALSE;
	garr_betriebsmeldungen[st_config_achse.i16_meld_startindex + 86] :=  FALSE;
	garr_betriebsmeldungen[st_config_achse.i16_meld_startindex + 87] :=  FALSE;
	garr_betriebsmeldungen[st_config_achse.i16_meld_startindex + 88] :=  FALSE;
	garr_betriebsmeldungen[st_config_achse.i16_meld_startindex + 89] :=  FALSE;
	garr_betriebsmeldungen[st_config_achse.i16_meld_startindex + 90] :=  FALSE;
	garr_betriebsmeldungen[st_config_achse.i16_meld_startindex + 91] :=  FALSE;
	garr_betriebsmeldungen[st_config_achse.i16_meld_startindex + 92] :=  FALSE;
	garr_betriebsmeldungen[st_config_achse.i16_meld_startindex + 93] :=  FALSE;
	garr_betriebsmeldungen[st_config_achse.i16_meld_startindex + 94] :=  FALSE;
	garr_betriebsmeldungen[st_config_achse.i16_meld_startindex + 95] :=  FALSE;
	garr_betriebsmeldungen[st_config_achse.i16_meld_startindex + 96] :=  FALSE;
	garr_betriebsmeldungen[st_config_achse.i16_meld_startindex + 97] :=  FALSE;
	garr_betriebsmeldungen[st_config_achse.i16_meld_startindex + 98] :=  FALSE;
	garr_betriebsmeldungen[st_config_achse.i16_meld_startindex + 99] :=  FALSE;
END_IF
END_PROGRAM

(* POU EPT Lib/Achsen/BECKHOFF/ST_AxisJobCtrl_Motion, ST *)
FUNCTION_BLOCK ST_AxisJobCtrl_Motion
VAR_INPUT
	e_referenznocken						: BOOL;
	b_refsensor_vorhanden				: BOOL;
	b_limitsensor_positiv_vorhanden		: BOOL;
	b_limitsensor_negativ_vorhanden		: BOOL;
	i16_achstyp							: enum_ecd_typ;
	lr_override_vorgabe					: LREAL;
	st_position							: struct_ecd_positionen;
	mc_richtung_modulo					: MC_Direction;
	mc_richtung_velocity					: MC_Direction;
											(*default: MC_Positive_Direction := 1,
											MC_Shortest_Way ,
									    		MC_Negative_Direction,
									    		MC_Current_Direction *)
	mc_referenzmodus 					: MC_HomingMode; (* default: MC_DefaultHoming   default homing as defined in the SystemManager encoder parameters *)
	mc_buffermode_axis					: MC_BufferMode;     (*	MC_Aborting,	->sofortiger Abbruch der momentanen Bewegung, bei einem neuen Verfahrbefehl
														MC_Buffered,
														MC_BlendingLow,
														MC_BlendingPrevious,
														MC_BlendingNext,
														MC_BlendingHigh *)
	ui16_soeparam_write_value				: UINT;
	w_idn								: WORD;
	i16_nc_parameter_nummer				: INT;
	r_wert_nc_write_parameter				: LREAL;
	st_vorgabe_geschwindigkeiten			: struct_ecd_geschwindigkeiten;
	lr_soll_geschwindigkeit					: LREAL;
	b_bedingung_sls						: BOOL;
	st_ads_info							: struct_ads_info;
	st_eccoe_sdo						: struct_eccoe_sdo;
	b_TriggerInput						: BOOL;
	b_FallingEdge						: BOOL;
END_VAR
VAR_OUTPUT
	ui16_soeparam_read_value			: UINT;
	r_wert_nc_read_parameter				: LREAL;
	lr_RecPos							: LREAL;
END_VAR
VAR_IN_OUT
	st_masterachse						: AXIS_REF;
	st_visu_axis							: struct_ecd_visu;
	st_ecd_cmd							: struct_ecd_cmd;
END_VAR
VAR
	fb_ton_cmd_timeout					: TON;
	t_cmd_timeout						: TIME;
	t_ads_timeout							: TIME;
	fb_ton_vz							: TON;
	b_jog_vorwaerts_execute				: BOOL := FALSE;
	b_jog_rueckwaerts_execute				: BOOL := FALSE;
	e_limit_sensor_positive				AT %I* : BOOL;
	e_limit_sensor_negative				AT %I* : BOOL;
	e_referenz_sensor						AT %I* : BOOL;
	fb_f_trig_limit_sensor_positiv			: F_TRIG;
	fb_f_trig_limit_sensor_negativ			: F_TRIG;
	fb_cmd_history						: ST_CommandHistory;

	mc_power_axis 						: MC_Power;
	mc_reset_axis						: MC_Reset;
	mc_home_axis 						: MC_Home;
	mc_setposition_axis					: MC_SetPosition;
	mc_jog_axis							: MC_Jog;
	mc_moveabsolute_axis 				: MC_MoveAbsolute;
	mc_moveabsolutenext_axis 			: MC_MoveAbsolute;
	mc_moverelative_axis 					: MC_MoveRelative;
	mc_movevelocity_axis 					: MC_MoveVelocity;
	mc_movemodulo_axis					: MC_MoveModulo;
	mc_stop_axis 						: MC_Stop;
	mc_halt_axis							: MC_Halt;
	mc_touch_probe					: MC_TouchProbe;
	mc_abort_trigger						: MC_AbortTrigger;
	TriggerInput							:TRIGGER_REF;
	err_id								: DWORD := 0;
	fb_state_entry							: ST_StateEntry;
	fb_soe_reset							: FB_SoEReset;
	fb_soe_write							: FB_SoEWrite;
	fb_soe_read							: FB_SoERead;
	fb_ec_coe_sdo_write_ex				: FB_EcCoESdoWriteEx;
	fb_ec_coe_sdo_read_ex				: FB_EcCoESdoReadEx;
	mc_write_nc_parameter				: MC_WriteParameter;
	mc_read_nc_parameter				: MC_ReadParameter;
	fb_ads_write							: ADSWRITE;
	fb_ads_read							: ADSREAD;
	lr_override							: LREAL := 0.0;
	lr_override_reduziert					: LREAL := 0.0;
	lr_reduktionsfaktor						: LREAL := 5.0;
	lr_hm_master_act_velo					: LREAL := 0.0;
	lr_sollgeschwindigkeit					: LREAL := 0.0;
END_VAR
sub_TouchProbe();
(* Zeiten *)
fb_ton_cmd_timeout(IN:= , PT:=t_cmd_timeout, Q=> , ET=> );
fb_ton_vz(IN:= , PT:= , Q=> , ET=> );

(* Flanken *)
fb_f_trig_limit_sensor_positiv(CLK:= e_limit_sensor_positive, Q=> );
fb_f_trig_limit_sensor_negativ(CLK:= e_limit_sensor_negative, Q=> );

(* =====Beschränkung des Overrides wegen SLS bei offenen Türen===== *)
IF b_bedingung_sls THEN
	IF i16_achstyp = RUND OR  i16_achstyp = RUND_VIRTUELL THEN
		lr_hm_master_act_velo := st_masterachse.NcToPlc.ActVelo * 60 / 360;
	ELSE
		lr_hm_master_act_velo := st_masterachse.NcToPlc.ActVelo;
	END_IF
	IF ABS(lr_hm_master_act_velo) < st_vorgabe_geschwindigkeiten.lr_jog THEN
		lr_override := lr_override_reduziert := lr_override_vorgabe;
	ELSE
		lr_override_reduziert := lr_override_reduziert - lr_reduktionsfaktor;
		IF lr_override_reduziert >= 0 OR lr_override_reduziert <= 100 THEN
			lr_override := lr_override_reduziert;
		END_IF
	END_IF
ELSE
	lr_override := lr_override_vorgabe;
END_IF

(* =====Beschränkung der Achsgeschwindigkeiten===== *)
(* Verrechnet nach Rund/Linear wird weiter unten *)
lr_sollgeschwindigkeit := lr_soll_geschwindigkeit;

(* Beschränkung der Geschwindigkeit *)
IF lr_sollgeschwindigkeit > st_vorgabe_geschwindigkeiten.lr_auto_max THEN
	lr_sollgeschwindigkeit := st_vorgabe_geschwindigkeiten.lr_auto_max;
ELSIF lr_sollgeschwindigkeit < st_vorgabe_geschwindigkeiten.lr_auto_min THEN
	lr_sollgeschwindigkeit := st_vorgabe_geschwindigkeiten.lr_auto_min ;
END_IF

(* ======Ausgabe von Position und Geschwindigkeit der Achse===== *)
IF i16_achstyp = RUND OR  i16_achstyp = RUND_VIRTUELL THEN
	(* INT-Daten *)
	IF LREAL_TO_DINT(st_masterachse.NcToPlc.ModuloActPos) = 360 THEN
		st_visu_axis.i32_position_ist := 0;
	ELSE
		st_visu_axis.i32_position_ist := LREAL_TO_DINT(st_masterachse.NcToPlc.ModuloActPos);
	END_IF
	st_visu_axis.i32_geschwindigkeit_ist := LREAL_TO_DINT(st_masterachse.NcToPlc.ActVelo * 60 / 360); (* Hub = Grad/sec / 360 * 60s *)

	(* LREAL-DATEN *)
	st_visu_axis.lr_position_ist :=st_masterachse.NcToPlc.ModuloActPos;
	st_visu_axis.lr_geschwindigkeit_ist := st_masterachse.NcToPlc.ActVelo * 60 / 360; (* Hub = Grad/sec / 360 * 60s *)
ELSIF i16_achstyp = LINEAR OR i16_achstyp = LINEAR_VIRTUELL THEN
	st_visu_axis.lr_position_ist :=st_masterachse.NcToPlc.ActPos;
	st_visu_axis.lr_geschwindigkeit_ist := st_masterachse.NcToPlc.ActVelo;
ELSE
	st_visu_axis.lr_position_ist :=st_masterachse.NcToPlc.ActPos;
	st_visu_axis.lr_geschwindigkeit_ist := st_masterachse.NcToPlc.ActVelo;
END_IF

(* ======================================Schrittkette Drivebefehle======================================== *)
fb_state_entry(
	i16_next_step:= , 
	i16_pos:= 1,
	s_debugtext:= ,
	E=> ,
	X=> ,
	i16_step=> ,
	i16_last_step=> );

CASE fb_state_entry.i16_step OF
(*=======================================================*)
	0:	(* Init *)
		st_ecd_cmd.b_job_fehler := FALSE;
		st_ecd_cmd.enu_cmd := NO_COMMAND;
		mc_buffermode_axis := MC_Aborting;
		t_cmd_timeout := T#10s;
		t_ads_timeout := t#10s;
		err_id :=0;

		b_jog_vorwaerts_execute := FALSE;
		b_jog_rueckwaerts_execute := FALSE;
		mc_power_axis.Enable := FALSE;
		mc_reset_axis.Execute := FALSE;
		mc_home_axis.Execute := FALSE;
		mc_moveabsolute_axis.Execute := FALSE;
		mc_moverelative_axis.Execute := FALSE;
		mc_movevelocity_axis.Execute := FALSE;
		mc_movemodulo_axis.Execute := FALSE;
		mc_setposition_axis.Execute := FALSE;
		mc_halt_axis.Execute := FALSE;
		mc_stop_axis.Execute := FALSE;
		mc_touch_probe.Execute := FALSE;
		fb_soe_reset.Execute := FALSE;
		fb_soe_write.Execute := FALSE;
		fb_soe_read.Execute := FALSE;
		fb_ec_coe_sdo_write_ex.bExecute := FALSE;
		fb_ec_coe_sdo_write_ex.bExecute := FALSE;
		mc_write_nc_parameter.Execute := FALSE;
		mc_read_nc_parameter.Enable := FALSE;
		fb_ads_write.WRITE := FALSE;
		fb_ads_read.READ := FALSE;

		st_ecd_cmd.meldungen.sm_power_enable := FALSE;
		st_ecd_cmd.meldungen.sm_power_disable := FALSE;
		st_ecd_cmd.meldungen.sm_reset := FALSE;
		st_ecd_cmd.meldungen.sm_home := FALSE;
		st_ecd_cmd.meldungen.sm_setposition := FALSE;
		st_ecd_cmd.meldungen.sm_jog_vorwaerts := FALSE;
		st_ecd_cmd.meldungen.sm_jog_rueckwaerts := FALSE;
		st_ecd_cmd.meldungen.sm_move_absolute := FALSE;
		st_ecd_cmd.meldungen.sm_move_relative := FALSE;
		st_ecd_cmd.meldungen.sm_move_velocity := FALSE;
		st_ecd_cmd.meldungen.sm_move_modulo := FALSE;
		st_ecd_cmd.meldungen.sm_stop_axis := FALSE;
		st_ecd_cmd.meldungen.sm_halt_axis := FALSE;
		st_ecd_cmd.meldungen.sm_motion_command_timeout := FALSE;
		st_ecd_cmd.meldungen.sm_limit_positiv_erreicht := FALSE;
		st_ecd_cmd.meldungen.sm_limit_negativ_erreicht := FALSE;
		st_ecd_cmd.meldungen.sm_write_soe_parameter := FALSE;
		st_ecd_cmd.meldungen.sm_read_soe_parameter := FALSE;
		st_ecd_cmd.meldungen.sm_write_nc_parameter := FALSE;
		st_ecd_cmd.meldungen.sm_read_nc_parameter := FALSE;
		st_ecd_cmd.meldungen.sm_write_ads_parameter := FALSE;
		st_ecd_cmd.meldungen.sm_read_ads_parameter := FALSE;
		st_ecd_cmd.meldungen.sm_ec_coe_sdo_write_ex := FALSE;
		st_ecd_cmd.meldungen.sm_ec_coe_sdo_read_ex := FALSE;
		st_ecd_cmd.meldungen.sm_touch_probe_defect := FALSE;
		st_ecd_cmd.meldungen.sm_touch_probe_err := FALSE;
		fb_state_entry.i16_next_step := 1;

